C09096=1089.886,417.075,-101.948,178.028,26.123,154.162
C09097=1089.893,417.322,-101.988,178.031,26.132,154.164
C09098=1089.899,417.568,-102.030,178.035,26.142,154.166
C09099=1089.905,417.814,-102.071,178.038,26.152,154.168
C09100=1089.912,418.061,-102.112,178.042,26.162,154.170
C09101=1089.918,418.307,-102.154,178.045,26.171,154.172
C09102=1089.925,418.554,-102.196,178.048,26.181,154.174
C09103=1089.931,418.800,-102.237,178.051,26.191,154.176
C09104=1089.938,419.047,-102.278,178.055,26.201,154.179
C09105=1089.944,419.293,-102.320,178.058,26.211,154.180
C09106=1089.950,419.539,-102.361,178.062,26.221,154.183
C09107=1089.956,419.786,-102.403,178.065,26.231,154.185
C09108=1089.962,420.032,-102.444,178.069,26.241,154.187
C09109=1089.970,420.279,-102.486,178.072,26.251,154.189
C09110=1089.976,420.525,-102.527,178.075,26.261,154.191
C09111=1089.982,420.772,-102.570,178.078,26.271,154.193
C09112=1089.988,421.018,-102.611,178.082,26.281,154.195
C09113=1089.995,421.265,-102.653,178.086,26.291,154.197
C09114=1090.001,421.512,-102.695,178.089,26.302,154.200
C09115=1090.008,421.757,-102.736,178.092,26.312,154.202
C09116=1090.015,422.004,-102.778,178.096,26.322,154.204
C09117=1090.021,422.250,-102.820,178.099,26.332,154.206
C09118=1090.027,422.497,-102.861,178.103,26.343,154.208
C09119=1090.034,422.742,-102.904,178.106,26.353,154.210
C09120=1090.040,422.989,-102.945,178.110,26.364,154.213
C09121=1090.047,423.236,-102.988,178.113,26.374,154.215
C09122=1090.053,423.482,-103.029,178.117,26.385,154.217
C09123=1090.060,423.728,-103.072,178.120,26.395,154.219
C09124=1090.066,423.974,-103.113,178.124,26.406,154.221
C09125=1090.073,424.221,-103.156,178.127,26.417,154.224
C09126=1090.079,424.454,-103.196,178.130,26.427,154.226
C09127=1090.085,424.688,-103.235,178.133,26.437,154.228
C09128=1090.090,424.922,-103.276,178.137,26.447,154.230
C09129=1090.097,425.156,-103.316,178.140,26.457,154.232
C09130=1090.103,425.389,-103.356,178.144,26.467,154.235
C09131=1090.109,425.623,-103.396,178.146,26.478,154.237
C09132=1090.115,425.857,-103.436,178.150,26.488,154.239
C09133=1090.122,426.091,-103.477,178.153,26.498,154.241
C09134=1090.128,426.336,-103.519,178.157,26.509,154.244
C09135=1090.135,426.583,-103.561,178.160,26.520,154.246
C09136=1090.141,426.830,-103.604,178.163,26.531,154.248
C09137=1090.148,427.076,-103.646,178.168,26.542,154.251
C09138=1090.154,427.322,-103.688,178.171,26.553,154.253
C09139=1090.161,427.568,-103.731,178.174,26.564,154.255
C09140=1090.167,427.814,-103.774,178.178,26.575,154.258
C09141=1090.174,428.061,-103.816,178.181,26.587,154.260
C09142=1090.180,428.307,-103.859,178.185,26.597,154.262
C09143=1090.187,428.553,-103.901,178.188,26.609,154.265
C09144=1090.194,428.799,-103.944,178.192,26.620,154.267
C09145=1090.200,429.045,-103.986,178.196,26.631,154.270
C09146=1090.207,429.292,-104.030,178.199,26.643,154.272
C09147=1090.213,429.538,-104.072,178.202,26.654,154.275
C09148=1090.219,429.783,-104.116,178.206,26.665,154.277
C09149=1090.226,430.030,-104.158,178.210,26.677,154.280
C09150=1090.233,430.276,-104.201,178.213,26.688,154.282
C09151=1090.239,430.523,-104.244,178.216,26.700,154.285
C09152=1090.246,430.769,-104.286,178.220,26.712,154.287
C09153=1090.252,431.015,-104.330,178.224,26.724,154.290
C09154=1090.259,431.261,-104.373,178.227,26.735,154.292
C09155=1090.265,431.507,-104.415,178.231,26.747,154.295
C09156=1090.272,431.753,-104.459,178.235,26.759,154.297
C09157=1090.279,431.999,-104.501,178.238,26.770,154.300
C09158=1090.285,432.245,-104.545,178.241,26.782,154.302
C09159=1090.292,432.491,-104.588,178.245,26.794,154.305
C09160=1090.298,432.737,-104.632,178.249,26.806,154.308
C09161=1090.305,432.983,-104.674,178.252,26.818,154.310
C09162=1090.312,433.229,-104.718,178.255,26.830,154.313
C09163=1090.318,433.476,-104.761,178.260,26.842,154.316
C09164=1090.325,433.722,-104.804,178.263,26.854,154.318
C09165=1090.331,433.968,-104.848,178.267,26.866,154.321
C09166=1090.338,434.214,-104.891,178.270,26.879,154.324
C09167=1090.345,434.460,-104.935,178.274,26.890,154.326
C09168=1090.351,434.706,-104.978,178.278,26.903,154.329
C09169=1090.358,434.952,-105.022,178.281,26.915,154.332
C09170=1090.364,435.198,-105.065,178.284,26.927,154.334
C09171=1090.371,435.444,-105.109,178.288,26.940,154.337
C09172=1090.377,435.690,-105.153,178.292,26.952,154.340
C09173=1090.384,435.936,-105.196,178.296,26.965,154.343
C09174=1090.391,436.182,-105.240,178.299,26.977,154.345
C09175=1090.397,436.428,-105.283,178.303,26.990,154.348
C09176=1090.404,436.674,-105.327,178.306,27.002,154.351
C09177=1090.411,436.920,-105.371,178.310,27.015,154.354
C09178=1090.418,437.166,-105.415,178.314,27.028,154.356
C09179=1090.424,437.412,-105.459,178.318,27.041,154.359
C09180=1090.431,437.658,-105.503,178.321,27.053,154.362
C09181=1090.438,437.904,-105.546,178.325,27.066,154.365
C09182=1090.448,438.250,-105.608,178.330,27.084,154.369
C09183=1090.457,438.596,-105.669,178.335,27.102,154.373
C09184=1090.466,438.942,-105.732,178.340,27.121,154.377
C09185=1090.475,439.288,-105.794,178.345,27.139,154.381
C09186=1090.482,439.534,-105.838,178.349,27.152,154.384
C09187=1090.490,439.780,-105.882,178.353,27.165,154.387
C09188=1090.496,440.026,-105.926,178.356,27.178,154.390
C09189=1090.503,440.271,-105.970,178.361,27.192,154.393
C09190=1090.510,440.518,-106.015,178.364,27.205,154.396
C09191=1090.517,440.763,-106.059,178.368,27.219,154.399
C09192=1090.523,441.009,-106.103,178.372,27.232,154.402
C09193=1090.530,441.255,-106.148,178.375,27.245,154.405
C09194=1090.537,441.501,-106.192,178.379,27.259,154.408
C09195=1090.544,441.747,-106.236,178.383,27.273,154.411
C09196=1090.550,441.992,-106.281,178.386,27.286,154.414
C09197=1090.557,442.239,-106.325,178.390,27.300,154.417
C09198=1090.563,442.485,-106.370,178.394,27.313,154.420
C09199=1090.570,442.730,-106.415,178.397,27.327,154.423
C09200=1090.578,442.976,-106.460,178.401,27.341,154.427
C09201=1090.584,443.222,-106.504,178.406,27.355,154.430
C09202=1090.591,443.467,-106.548,178.410,27.369,154.433
C09203=1090.598,443.713,-106.593,178.413,27.383,154.436
C09204=1090.604,443.959,-106.638,178.417,27.397,154.439
C09205=1090.611,444.205,-106.683,178.421,27.411,154.442
C09206=1090.618,444.450,-106.728,178.425,27.425,154.446
C09207=1090.625,444.696,-106.773,178.428,27.439,154.449
C09208=1090.632,444.942,-106.817,178.431,27.453,154.452
C09209=1090.639,445.188,-106.863,178.435,27.468,154.455
C09210=1090.645,445.434,-106.907,178.438,27.481,154.459
C09211=1090.653,445.680,-106.952,178.440,27.495,154.462
C09212=1090.659,445.925,-106.997,178.443,27.509,154.465
C09213=1090.666,446.171,-107.042,178.445,27.524,154.469
C09214=1090.673,446.416,-107.088,178.447,27.538,154.472
C09215=1090.680,446.662,-107.133,178.449,27.552,154.475
C09216=1090.686,446.908,-107.178,178.452,27.566,154.479
C09217=1090.694,447.154,-107.223,178.454,27.580,154.482
C09218=1090.700,447.399,-107.269,178.455,27.593,154.485
C09219=1090.707,447.645,-107.313,178.456,27.608,154.489
C09220=1090.714,447.891,-107.359,178.458,27.622,154.492
C09221=1090.721,448.137,-107.404,178.458,27.635,154.496
C09222=1090.728,448.382,-107.450,178.459,27.649,154.499
C09223=1090.735,448.628,-107.495,178.461,27.663,154.503
C09224=1090.742,448.873,-107.540,178.461,27.677,154.506
C09225=1090.749,449.119,-107.586,178.462,27.691,154.510
C09226=1090.756,449.364,-107.631,178.462,27.705,154.513
C09227=1090.763,449.610,-107.676,178.462,27.719,154.517
C09228=1090.770,449.855,-107.721,178.463,27.732,154.520
C09229=1090.780,450.102,-107.765,178.462,27.745,154.523
C09230=1090.397,450.093,-107.952,178.418,27.943,154.578
C09231=1090.387,449.848,-107.908,178.417,27.930,154.575
C09232=1090.380,449.603,-107.862,178.417,27.917,154.571
C09233=1090.372,449.358,-107.817,178.417,27.903,154.568
C09234=1090.366,449.112,-107.771,178.416,27.889,154.564
C09235=1090.359,448.867,-107.726,178.416,27.875,154.561
C09236=1090.352,448.620,-107.680,178.415,27.861,154.557
C09237=1090.344,448.375,-107.635,178.415,27.847,154.554
C09238=1090.338,448.129,-107.590,178.413,27.833,154.550
C09239=1090.331,447.884,-107.544,178.412,27.819,154.547
C09240=1090.323,447.638,-107.499,178.411,27.805,154.543
C09241=1090.317,447.392,-107.454,178.410,27.791,154.540
C09242=1090.310,447.147,-107.408,178.407,27.777,154.537
C09243=1090.303,446.900,-107.363,178.406,27.763,154.533
C09244=1090.297,446.655,-107.318,178.404,27.749,154.530
C09245=1090.290,446.409,-107.272,178.402,27.735,154.526
C09246=1090.282,446.163,-107.227,178.399,27.721,154.523
C09247=1090.276,445.918,-107.182,178.396,27.706,154.520
C09248=1090.269,445.672,-107.137,178.394,27.692,154.516
C09249=1090.262,445.427,-107.092,178.391,27.678,154.513
C09250=1090.255,445.181,-107.047,178.388,27.664,154.510
C09251=1090.249,444.935,-107.001,178.385,27.650,154.506
C09252=1090.241,444.689,-106.957,178.380,27.636,154.503
C09253=1090.235,444.444,-106.912,178.377,27.622,154.500
C09254=1090.227,444.198,-106.867,178.373,27.607,154.497
C09255=1090.220,443.952,-106.822,178.369,27.593,154.494
C09256=1090.214,443.706,-106.777,178.366,27.580,154.490
C09257=1090.207,443.461,-106.732,178.362,27.565,154.487
C09258=1090.200,443.214,-106.687,178.358,27.551,154.484
C09259=1090.193,442.969,-106.643,178.353,27.537,154.481
C09260=1090.186,442.724,-106.598,178.350,27.524,154.478
C09261=1090.179,442.477,-106.554,178.346,27.510,154.475
C09262=1090.173,442.231,-106.509,178.342,27.496,154.472
C09263=1090.166,441.985,-106.464,178.339,27.482,154.468
C09264=1090.159,441.740,-106.419,178.335,27.468,154.465
C09265=1090.153,441.494,-106.376,178.330,27.455,154.462
C09266=1090.146,441.248,-106.331,178.327,27.442,154.459
C09267=1090.139,441.003,-106.286,178.323,27.428,154.456
C09268=1090.132,440.757,-106.242,178.320,27.415,154.453
C09269=1090.125,440.511,-106.197,178.316,27.401,154.450
C09270=1090.119,440.265,-106.153,178.312,27.387,154.447
C09271=1090.112,440.019,-106.109,178.308,27.374,154.444
C09272=1090.105,439.773,-106.065,178.304,27.361,154.441
C09273=1090.099,439.544,-106.024,178.301,27.349,154.439
C09274=1090.092,439.316,-105.982,178.297,27.337,154.436
C09275=1090.086,439.088,-105.942,178.294,27.325,154.433
C09276=1090.080,438.860,-105.901,178.290,27.312,154.430
C09277=1090.073,438.631,-105.860,178.287,27.300,154.428
C09278=1090.067,438.403,-105.819,178.284,27.288,154.425
C09279=1090.060,438.174,-105.777,178.280,27.276,154.422
C09280=1090.054,437.945,-105.738,178.276,27.264,154.420
C09281=1090.047,437.700,-105.693,178.272,27.251,154.417
C09282=1090.041,437.454,-105.649,178.268,27.238,154.414
C09283=1090.034,437.208,-105.605,178.265,27.226,154.411
C09284=1090.027,436.962,-105.562,178.262,27.213,154.408
C09285=1090.020,436.716,-105.518,178.257,27.200,154.405
C09286=1090.014,436.470,-105.474,178.254,27.188,154.403
C09287=1090.007,436.224,-105.430,178.250,27.175,154.400
C09288=1090.001,435.978,-105.386,178.247,27.163,154.397
C09289=1089.994,435.732,-105.343,178.242,27.150,154.394
C09290=1089.987,435.486,-105.299,178.239,27.138,154.392
C09291=1089.981,435.240,-105.255,178.235,27.125,154.389
C09292=1089.974,434.994,-105.212,178.231,27.113,154.386
C09293=1089.967,434.749,-105.168,178.228,27.101,154.383
C09294=1089.960,434.502,-105.124,178.224,27.088,154.381
C09295=1089.954,434.255,-105.081,178.221,27.076,154.378
C09296=1089.948,434.010,-105.038,178.217,27.064,154.375
C09297=1089.941,433.764,-104.994,178.213,27.051,154.373
C09298=1089.934,433.518,-104.950,178.210,27.039,154.370
C09299=1089.928,433.272,-104.908,178.206,27.027,154.367
C09300=1089.922,433.026,-104.864,178.202,27.015,154.365
C09301=1089.915,432.780,-104.821,178.199,27.003,154.362
C09302=1089.908,432.534,-104.778,178.195,26.991,154.359
C09303=1089.901,432.288,-104.734,178.191,26.979,154.357
C09304=1089.895,432.042,-104.691,178.188,26.967,154.354
C09305=1089.888,431.796,-104.648,178.184,26.956,154.352
C09306=1089.882,431.549,-104.605,178.180,26.943,154.349
C09307=1089.875,431.303,-104.562,178.177,26.932,154.347
C09308=1089.868,431.057,-104.518,178.173,26.920,154.344
C09309=1089.862,430.811,-104.476,178.170,26.909,154.341
C09310=1089.855,430.565,-104.432,178.165,26.897,154.339
C09311=1089.848,430.318,-104.389,178.162,26.885,154.336
C09312=1089.841,430.072,-104.347,178.159,26.874,154.334
C09313=1089.835,429.826,-104.304,178.155,26.862,154.331
C09314=1089.828,429.580,-104.261,178.151,26.851,154.329
C09315=1089.823,429.334,-104.218,178.148,26.839,154.326
C09316=1089.816,429.088,-104.175,178.144,26.828,154.324
C09317=1089.809,428.841,-104.133,178.141,26.816,154.321
C09318=1089.803,428.595,-104.090,178.137,26.805,154.319
C09319=1089.796,428.349,-104.047,178.134,26.794,154.317
C09320=1089.789,428.102,-104.004,178.130,26.782,154.314
C09321=1089.783,427.857,-103.962,178.126,26.771,154.312
C09322=1089.776,427.610,-103.920,178.123,26.760,154.309
C09323=1089.770,427.364,-103.877,178.119,26.749,154.307
C09324=1089.763,427.118,-103.834,178.116,26.738,154.305
C09325=1089.756,426.871,-103.792,178.112,26.727,154.302
C09326=1089.750,426.626,-103.749,178.109,26.716,154.300
C09327=1089.743,426.379,-103.707,178.105,26.705,154.298
C09328=1089.736,426.133,-103.664,178.101,26.694,154.295
C09329=1089.731,425.899,-103.623,178.098,26.684,154.293
C09330=1089.724,425.665,-103.584,178.095,26.673,154.291
C09331=1089.717,425.430,-103.543,178.091,26.663,154.289
C09332=1089.712,425.196,-103.503,178.088,26.653,154.286
C09333=1089.705,424.962,-103.462,178.085,26.643,154.284
C09334=1089.699,424.728,-103.423,178.081,26.632,154.282
C09335=1089.694,424.493,-103.382,178.078,26.622,154.280
C09336=1089.687,424.260,-103.342,178.074,26.612,154.278
C09337=1089.681,424.013,-103.300,178.071,26.601,154.275
C09338=1089.674,423.766,-103.258,178.067,26.591,154.273
C09339=1089.668,423.520,-103.216,178.064,26.580,154.271
C09340=1089.661,423.274,-103.174,178.060,26.569,154.269
C09341=1089.655,423.028,-103.132,178.057,26.559,154.266
C09342=1089.648,422.781,-103.090,178.053,26.548,154.264
C09343=1089.642,422.535,-103.048,178.050,26.538,154.262
C09344=1089.635,422.289,-103.006,178.046,26.527,154.260
C09345=1089.629,422.042,-102.964,178.043,26.517,154.258
C09346=1089.623,421.796,-102.922,178.040,26.507,154.256
C09347=1089.616,421.550,-102.880,178.037,26.497,154.253
C09348=1089.609,421.303,-102.838,178.033,26.487,154.251
C09349=1089.604,421.056,-102.797,178.029,26.476,154.249
C09350=1089.597,420.810,-102.754,178.026,26.466,154.247
C09351=1089.590,420.564,-102.713,178.022,26.456,154.245
C09352=1089.583,420.317,-102.671,178.019,26.446,154.243
C09353=1089.577,420.071,-102.630,178.015,26.436,154.241
C09354=1089.571,419.824,-102.588,178.012,26.426,154.238
C09355=1089.565,419.578,-102.547,178.008,26.415,154.236
C09356=1089.557,419.332,-102.505,178.005,26.406,154.234
C09357=1089.551,419.086,-102.463,178.002,26.396,154.232
C09358=1089.545,418.839,-102.421,177.998,26.386,154.230
C09359=1089.539,418.593,-102.380,177.995,26.376,154.228
C09360=1089.532,418.346,-102.339,177.991,26.366,154.226
C09361=1089.526,418.100,-102.297,177.987,26.356,154.224
C09362=1089.519,417.853,-102.255,177.985,26.346,154.222
C09363=1089.513,417.607,-102.214,177.981,26.336,154.220
C09364=1089.507,417.360,-102.174,177.978,26.327,154.218
C09365=1089.500,417.113,-102.132,177.974,26.317,154.216
C09366=1089.494,416.867,-102.091,177.970,26.307,154.214
C09367=1089.488,416.621,-102.049,177.968,26.297,154.212
C09368=1089.481,416.374,-102.008,177.964,26.288,154.210
C09369=1089.475,416.128,-101.966,177.960,26.278,154.208
C09370=1089.469,415.881,-101.925,177.957,26.268,154.206
C09371=1089.462,415.635,-101.884,177.954,26.259,154.204
C09372=1089.456,415.389,-101.843,177.950,26.250,154.202
C09373=1089.449,415.141,-101.802,177.947,26.240,154.200
C09374=1089.443,414.895,-101.761,177.943,26.230,154.198
C09375=1089.436,414.649,-101.720,177.940,26.221,154.196
C09376=1089.430,414.402,-101.679,177.937,26.212,154.194
C09377=1089.424,414.156,-101.638,177.933,26.202,154.192
C09378=1089.417,413.909,-101.598,177.930,26.194,154.190
C09379=1089.411,413.662,-101.556,177.927,26.184,154.188
C09380=1089.404,413.416,-101.516,177.923,26.175,154.187
C09381=1089.398,413.169,-101.474,177.920,26.165,154.185
C09382=1089.391,412.923,-101.434,177.917,26.156,154.183
C09383=1089.386,412.676,-101.393,177.913,26.147,154.181
C09384=1089.379,412.430,-101.352,177.910,26.138,154.179
C09385=1089.374,412.202,-101.315,177.907,26.130,154.177
C09386=1089.367,411.976,-101.277,177.903,26.121,154.176
C09387=1089.362,411.749,-101.240,177.900,26.112,154.174
C09388=1089.355,411.522,-101.203,177.897,26.105,154.172
C09389=1089.350,411.296,-101.165,177.895,26.096,154.171
C09390=1089.344,411.069,-101.128,177.892,26.088,154.169
C09391=1089.339,410.843,-101.090,177.889,26.080,154.167
C09392=1089.332,410.616,-101.053,177.886,26.072,154.165
C09393=1089.326,410.369,-101.012,177.882,26.062,154.164
C09394=1089.320,410.123,-100.972,177.878,26.053,154.162
C09395=1089.314,409.876,-100.932,177.876,26.044,154.160
C09396=1089.308,409.630,-100.891,177.872,26.036,154.158
C09397=1089.302,409.383,-100.851,177.869,26.027,154.156
C09398=1089.295,409.136,-100.810,177.865,26.018,154.155
C09399=1089.288,408.889,-100.770,177.862,26.009,154.153
C09400=1089.282,408.643,-100.729,177.859,26.000,154.151
C09401=1089.276,408.396,-100.689,177.856,25.992,154.149
C09402=1089.270,408.149,-100.649,177.852,25.983,154.148
C09403=1089.264,407.903,-100.608,177.849,25.974,154.146
C09404=1089.258,407.656,-100.568,177.846,25.965,154.144
C09405=1089.251,407.410,-100.528,177.843,25.957,154.142
C09406=1089.245,407.163,-100.488,177.839,25.948,154.141
C09407=1089.239,406.917,-100.448,177.836,25.940,154.139
C09408=1089.233,406.670,-100.407,177.832,25.931,154.137
C09409=1089.227,406.423,-100.367,177.829,25.923,154.136
C09410=1089.220,406.176,-100.327,177.826,25.914,154.134
C09411=1089.214,405.930,-100.287,177.823,25.906,154.132
C09412=1089.208,405.683,-100.247,177.820,25.897,154.130
C09413=1089.201,405.437,-100.207,177.816,25.889,154.129
C09414=1089.195,405.189,-100.168,177.813,25.881,154.127
C09415=1089.189,404.943,-100.127,177.809,25.872,154.125
C09416=1089.183,404.696,-100.087,177.807,25.864,154.124
C09417=1089.176,404.449,-100.048,177.804,25.855,154.122
C09418=1089.170,404.203,-100.008,177.800,25.847,154.121
C09419=1089.164,403.956,-99.968,177.797,25.839,154.119
C09420=1089.158,403.709,-99.928,177.793,25.830,154.117
C09421=1089.151,403.463,-99.888,177.790,25.823,154.116
C09422=1089.145,403.215,-99.849,177.787,25.814,154.114
C09423=1089.139,402.969,-99.808,177.783,25.806,154.112
C09424=1089.133,402.722,-99.769,177.781,25.798,154.111
C09425=1089.126,402.475,-99.729,177.778,25.790,154.109
C09426=1089.120,402.228,-99.689,177.774,25.782,154.108
C09427=1089.113,401.982,-99.650,177.771,25.774,154.106
C09428=1089.107,401.735,-99.610,177.768,25.766,154.104
C09429=1089.101,401.488,-99.571,177.764,25.757,154.103
C09430=1089.095,401.242,-99.531,177.761,25.749,154.101
C09431=1089.089,400.995,-99.492,177.758,25.742,154.100
C09432=1089.083,400.748,-99.452,177.754,25.734,154.098
C09433=1089.077,400.501,-99.412,177.751,25.726,154.097
C09434=1089.070,400.254,-99.373,177.748,25.718,154.095
C09435=1089.064,400.007,-99.334,177.745,25.710,154.093
C09436=1089.058,399.761,-99.294,177.742,25.702,154.092
C09437=1089.052,399.514,-99.255,177.739,25.694,154.090
C09438=1089.046,399.267,-99.215,177.736,25.686,154.089
C09439=1089.039,399.020,-99.176,177.733,25.679,154.087
C09440=1089.034,398.774,-99.137,177.729,25.671,154.086
C09441=1089.028,398.547,-99.101,177.726,25.664,154.085
C09442=1089.022,398.321,-99.065,177.723,25.656,154.083
C09443=1089.016,398.095,-99.029,177.720,25.649,154.082
C09444=1089.010,397.869,-98.994,177.717,25.642,154.080
C09445=1089.005,397.643,-98.957,177.714,25.635,154.079
C09446=1088.998,397.417,-98.921,177.712,25.629,154.078
C09447=1088.994,397.191,-98.886,177.709,25.622,154.076
C09448=1088.987,396.964,-98.850,177.706,25.614,154.075
C09449=1088.982,396.718,-98.811,177.703,25.607,154.074
C09450=1088.976,396.471,-98.772,177.700,25.599,154.072
C09451=1088.969,396.224,-98.733,177.696,25.591,154.071
C09452=1088.964,395.977,-98.694,177.692,25.584,154.069
C09453=1088.957,395.730,-98.655,177.689,25.577,154.068
C09454=1088.951,395.483,-98.616,177.686,25.569,154.066
C09455=1088.945,395.237,-98.577,177.683,25.562,154.065
C09456=1088.938,394.990,-98.538,177.680,25.554,154.063
C09457=1088.932,394.743,-98.498,177.676,25.547,154.062
C09458=1088.926,394.496,-98.461,177.673,25.539,154.061
C09459=1088.920,394.249,-98.422,177.670,25.532,154.059
C09460=1088.914,394.003,-98.383,177.667,25.525,154.058
C09461=1088.907,393.756,-98.344,177.664,25.517,154.056
C09462=1088.902,393.508,-98.305,177.661,25.510,154.055
C09463=1088.895,393.262,-98.267,177.658,25.503,154.054
C09464=1088.889,393.015,-98.227,177.654,25.495,154.052
C09465=1088.883,392.768,-98.189,177.651,25.488,154.051
C09466=1088.877,392.522,-98.151,177.648,25.480,154.050
C09467=1088.871,392.275,-98.111,177.645,25.473,154.048
C09468=1088.865,392.028,-98.073,177.642,25.466,154.047
C09469=1088.859,391.781,-98.034,177.639,25.459,154.046
C09470=1088.853,391.534,-97.996,177.636,25.452,154.044
C09471=1088.846,391.287,-97.957,177.632,25.445,154.043
C09472=1088.840,391.040,-97.920,177.629,25.438,154.042
C09473=1088.833,390.793,-97.881,177.626,25.431,154.040
C09474=1088.828,390.546,-97.842,177.622,25.424,154.039
C09475=1088.821,390.299,-97.804,177.619,25.416,154.038
C09476=1088.815,390.053,-97.766,177.616,25.409,154.036
C09477=1088.808,389.806,-97.727,177.613,25.402,154.035
C09478=1088.802,389.559,-97.689,177.610,25.396,154.034
C09479=1088.797,389.311,-97.651,177.607,25.389,154.032
C09480=1088.790,389.065,-97.612,177.604,25.382,154.031
C09481=1088.785,388.819,-97.574,177.600,25.375,154.030
C09482=1088.778,388.571,-97.536,177.597,25.368,154.028
C09483=1088.772,388.325,-97.498,177.594,25.361,154.027
C09484=1088.765,388.078,-97.460,177.591,25.354,154.026
C09485=1088.759,387.831,-97.422,177.588,25.347,154.025
C09486=1088.754,387.583,-97.383,177.585,25.340,154.023
C09487=1088.747,387.337,-97.345,177.582,25.333,154.022
C09488=1088.742,387.090,-97.307,177.578,25.327,154.021
C09489=1088.735,386.843,-97.269,177.574,25.319,154.020
C09490=1088.729,386.596,-97.231,177.571,25.313,154.018
C09491=1088.723,386.349,-97.193,177.568,25.306,154.017
C09492=1088.717,386.102,-97.155,177.565,25.299,154.016
C09493=1088.711,385.855,-97.117,177.562,25.292,154.015
C09494=1088.705,385.608,-97.080,177.558,25.286,154.013
C09495=1088.698,385.361,-97.041,177.555,25.279,154.012
C09496=1088.692,385.115,-97.003,177.552,25.272,154.011
C09497=1088.687,384.895,-96.969,177.550,25.266,154.010
C09498=1088.682,384.676,-96.936,177.547,25.260,154.009
C09499=1088.676,384.457,-96.902,177.544,25.254,154.008
C09500=1088.671,384.237,-96.868,177.542,25.248,154.007
C09501=1088.666,384.018,-96.835,177.538,25.243,154.006
C09502=1088.660,383.798,-96.801,177.536,25.237,154.005
C09503=1088.655,383.578,-96.767,177.532,25.231,154.003
C09504=1088.650,383.360,-96.734,177.530,25.225,154.002
C09505=1088.644,383.112,-96.696,177.527,25.218,154.001
C09506=1088.638,382.865,-96.659,177.524,25.212,154.000
C09507=1088.632,382.618,-96.621,177.520,25.205,153.999
C09508=1088.626,382.371,-96.583,177.517,25.198,153.998
C09509=1088.620,382.124,-96.545,177.514,25.192,153.996
C09510=1088.613,381.877,-96.508,177.511,25.186,153.995
C09511=1088.607,381.630,-96.471,177.508,25.179,153.994
C09512=1088.602,381.383,-96.433,177.505,25.173,153.993
C09513=1088.596,381.137,-96.396,177.502,25.167,153.992
C09514=1088.589,380.889,-96.358,177.499,25.160,153.991
C09515=1088.583,380.642,-96.321,177.496,25.154,153.990
C09516=1088.577,380.395,-96.283,177.492,25.148,153.988
C09517=1088.571,380.148,-96.246,177.489,25.141,153.987
C09518=1088.565,379.901,-96.208,177.486,25.135,153.986
C09519=1088.558,379.654,-96.172,177.482,25.128,153.985
C09520=1088.553,379.407,-96.134,177.479,25.122,153.984
C09521=1088.547,379.160,-96.096,177.476,25.116,153.983
C09522=1088.540,378.913,-96.060,177.474,25.110,153.982
C09523=1088.534,378.666,-96.022,177.470,25.104,153.981
C09524=1088.529,378.419,-95.985,177.467,25.097,153.979
C09525=1088.522,378.171,-95.947,177.464,25.091,153.978
C09526=1088.516,377.924,-95.910,177.461,25.085,153.977
C09527=1088.510,377.677,-95.873,177.457,25.078,153.976
C09528=1088.504,377.430,-95.836,177.454,25.072,153.975
C09529=1088.498,377.183,-95.799,177.451,25.066,153.974
C09530=1088.492,376.936,-95.761,177.448,25.060,153.973
C09531=1088.487,376.689,-95.724,177.445,25.054,153.972
C09532=1088.480,376.442,-95.688,177.442,25.047,153.971
C09533=1088.474,376.195,-95.650,177.439,25.041,153.970
C09534=1088.469,375.948,-95.613,177.435,25.035,153.969
C09535=1088.462,375.701,-95.577,177.432,25.029,153.968
C09536=1088.457,375.454,-95.540,177.430,25.023,153.966
C09537=1088.450,375.207,-95.502,177.426,25.017,153.966
C09538=1088.445,374.960,-95.465,177.423,25.011,153.964
C09539=1088.439,374.712,-95.428,177.420,25.005,153.963
C09540=1088.433,374.465,-95.392,177.416,24.999,153.962
C09541=1088.427,374.218,-95.355,177.413,24.992,153.961
C09542=1088.421,373.971,-95.318,177.411,24.987,153.960
C09543=1088.415,373.724,-95.281,177.407,24.981,153.959
C09544=1088.408,373.477,-95.244,177.404,24.975,153.958
C09545=1088.402,373.229,-95.207,177.401,24.969,153.957
C09546=1088.396,372.982,-95.170,177.397,24.963,153.956
C09547=1088.390,372.735,-95.134,177.395,24.957,153.955
C09548=1088.384,372.488,-95.097,177.392,24.951,153.954
C09549=1088.378,372.241,-95.060,177.388,24.945,153.953
C09550=1088.372,371.993,-95.023,177.385,24.939,153.952
C09551=1088.366,371.746,-94.987,177.382,24.934,153.951
C09552=1088.360,371.500,-94.951,177.379,24.928,153.950
C09553=1088.350,371.088,-94.890,177.374,24.918,153.949
C09554=1088.340,370.677,-94.829,177.368,24.908,153.947
C09555=1088.330,370.266,-94.769,177.363,24.899,153.945
C09556=1088.320,369.855,-94.708,177.358,24.889,153.944
C09557=1088.315,369.608,-94.671,177.355,24.883,153.943
C09558=1088.308,369.361,-94.635,177.352,24.878,153.942
C09559=1088.302,369.113,-94.599,177.349,24.872,153.941
C09560=1088.297,368.866,-94.562,177.345,24.866,153.940
C09561=1088.290,368.619,-94.526,177.342,24.860,153.939
C09562=1088.284,368.371,-94.490,177.339,24.855,153.938
C09563=1088.278,368.124,-94.454,177.336,24.849,153.937
C09564=1088.272,367.877,-94.416,177.333,24.844,153.936
C09565=1088.267,367.630,-94.381,177.330,24.838,153.935
C09566=1088.261,367.383,-94.345,177.327,24.832,153.934
C09567=1088.254,367.136,-94.308,177.323,24.827,153.933
C09568=1088.249,366.888,-94.272,177.320,24.821,153.932
C09569=1088.243,366.641,-94.235,177.318,24.816,153.931
C09570=1088.237,366.394,-94.200,177.314,24.810,153.930
C09571=1088.231,366.147,-94.164,177.311,24.804,153.929
C09572=1088.226,365.899,-94.127,177.308,24.799,153.928
C09573=1088.219,365.652,-94.091,177.305,24.793,153.928
C09574=1088.213,365.404,-94.055,177.302,24.787,153.927
C09575=1088.207,365.158,-94.019,177.299,24.782,153.926
C09576=1088.201,364.910,-93.983,177.296,24.776,153.925
C09577=1088.195,364.663,-93.947,177.292,24.771,153.924
C09578=1088.189,364.415,-93.911,177.290,24.766,153.923
C09579=1088.183,364.168,-93.875,177.286,24.760,153.922
C09580=1088.177,363.921,-93.839,177.283,24.755,153.921
C09581=1088.171,363.674,-93.804,177.280,24.749,153.920
C09582=1088.165,363.426,-93.768,177.277,24.743,153.919
C09583=1088.159,363.179,-93.731,177.273,24.738,153.919
C09584=1088.154,362.932,-93.696,177.271,24.733,153.918
C09585=1088.147,362.684,-93.660,177.267,24.727,153.917
C09586=1088.141,362.437,-93.625,177.264,24.722,153.916
C09587=1088.135,362.190,-93.588,177.261,24.717,153.915
C09588=1088.130,361.943,-93.553,177.258,24.711,153.914
C09589=1088.124,361.695,-93.517,177.255,24.706,153.913
C09590=1088.118,361.447,-93.481,177.252,24.701,153.913
C09591=1088.112,361.200,-93.446,177.248,24.695,153.912
C09592=1088.106,360.953,-93.410,177.245,24.690,153.911
C09593=1088.100,360.705,-93.374,177.242,24.685,153.910
C09594=1088.094,360.458,-93.338,177.239,24.679,153.909
C09595=1088.088,360.211,-93.303,177.236,24.674,153.908
C09596=1088.082,359.963,-93.267,177.233,24.669,153.907
C09597=1088.076,359.715,-93.231,177.229,24.663,153.907
C09598=1088.070,359.469,-93.197,177.227,24.658,153.906
C09599=1088.064,359.221,-93.161,177.223,24.653,153.905
C09600=1088.058,358.973,-93.125,177.221,24.648,153.904
C09601=1088.053,358.727,-93.090,177.217,24.643,153.903
C09602=1088.046,358.479,-93.055,177.214,24.638,153.902
C09603=1088.040,358.231,-93.019,177.211,24.633,153.902
C09604=1088.034,357.984,-92.983,177.208,24.627,153.901
C09605=1088.025,357.589,-92.927,177.203,24.619,153.899
C09606=1088.015,357.193,-92.871,177.198,24.611,153.898
C09607=1088.006,356.798,-92.814,177.193,24.602,153.897
C09608=1087.997,356.402,-92.758,177.188,24.594,153.896
C09609=1087.990,356.155,-92.723,177.185,24.589,153.895
C09610=1087.985,355.908,-92.688,177.182,24.584,153.894
C09611=1087.979,355.660,-92.652,177.179,24.579,153.893
C09612=1087.972,355.412,-92.617,177.176,24.574,153.892
C09613=1087.967,355.165,-92.582,177.172,24.569,153.892
C09614=1087.961,354.918,-92.546,177.170,24.564,153.891
C09615=1087.956,354.670,-92.512,177.166,24.559,153.890
C09616=1087.949,354.423,-92.477,177.163,24.553,153.889
C09617=1087.944,354.176,-92.441,177.160,24.549,153.889
C09618=1087.938,353.928,-92.406,177.157,24.544,153.888
C09619=1087.932,353.681,-92.371,177.154,24.539,153.887
C09620=1087.926,353.433,-92.336,177.150,24.534,153.886
C09621=1087.920,353.186,-92.302,177.148,24.529,153.885
C09622=1087.914,352.938,-92.266,177.144,24.523,153.885
C09623=1087.909,352.691,-92.231,177.142,24.519,153.884
C09624=1087.902,352.443,-92.196,177.138,24.514,153.883
C09625=1087.897,352.196,-92.161,177.135,24.509,153.882
C09626=1087.890,351.948,-92.126,177.132,24.504,153.882
C09627=1087.885,351.701,-92.092,177.129,24.499,153.881
C09628=1087.878,351.453,-92.057,177.126,24.494,153.880
C09629=1087.873,351.206,-92.022,177.123,24.490,153.879
C09630=1087.867,350.958,-91.987,177.120,24.484,153.879
C09631=1087.860,350.711,-91.953,177.117,24.480,153.878
C09632=1087.855,350.464,-91.918,177.113,24.475,153.877
C09633=1087.849,350.216,-91.884,177.111,24.470,153.876
C09634=1087.843,349.969,-91.848,177.107,24.465,153.876
C09635=1087.837,349.721,-91.814,177.105,24.460,153.875
C09636=1087.832,349.473,-91.779,177.101,24.455,153.874
C09637=1087.825,349.226,-91.744,177.098,24.451,153.874
C09638=1087.820,348.978,-91.709,177.095,24.445,153.873
C09639=1087.814,348.731,-91.675,177.092,24.441,153.872
C09640=1087.808,348.483,-91.641,177.088,24.436,153.871
C09641=1087.802,348.236,-91.606,177.086,24.432,153.871
C09642=1087.796,347.989,-91.572,177.082,24.426,153.870
C09643=1087.790,347.741,-91.537,177.080,24.422,153.869
C09644=1087.785,347.493,-91.502,177.076,24.417,153.869
C09645=1087.778,347.245,-91.468,177.073,24.412,153.868
C09646=1087.772,346.998,-91.434,177.071,24.408,153.867
C09647=1087.767,346.751,-91.399,177.067,24.403,153.866
C09648=1087.761,346.503,-91.364,177.064,24.398,153.866
C09649=1087.755,346.255,-91.330,177.061,24.393,153.865
C09650=1087.750,346.008,-91.296,177.058,24.389,153.864
C09651=1087.743,345.760,-91.261,177.054,24.384,153.864
C09652=1087.737,345.513,-91.227,177.052,24.379,153.863
C09653=1087.732,345.265,-91.192,177.048,24.374,153.862
C09654=1087.726,345.018,-91.158,177.045,24.370,153.862
C09655=1087.720,344.770,-91.124,177.043,24.365,153.861
C09656=1087.714,344.522,-91.090,177.039,24.361,153.860
C09657=1087.705,344.129,-91.035,177.034,24.353,153.859
C09658=1087.696,343.737,-90.982,177.029,24.346,153.858
C09659=1087.686,343.344,-90.928,177.024,24.339,153.857
C09660=1087.676,342.952,-90.873,177.020,24.332,153.856
C09661=1087.671,342.704,-90.840,177.017,24.327,153.855
C09662=1087.666,342.456,-90.805,177.013,24.322,153.855
C09663=1087.659,342.208,-90.771,177.011,24.318,153.854
C09664=1087.653,341.961,-90.737,177.008,24.314,153.853
C09665=1087.647,341.714,-90.703,177.004,24.309,153.853
C09666=1087.642,341.466,-90.669,177.001,24.304,153.852
C09667=1087.635,341.218,-90.635,176.998,24.299,153.851
C09668=1087.629,340.971,-90.601,176.995,24.295,153.851
C09669=1087.624,340.723,-90.568,176.992,24.291,153.850
C09670=1087.618,340.475,-90.533,176.989,24.286,153.849
C09671=1087.612,340.228,-90.499,176.986,24.281,153.849
C09672=1087.606,339.979,-90.466,176.983,24.277,153.848
C09673=1087.600,339.732,-90.432,176.980,24.272,153.848
C09674=1087.594,339.485,-90.398,176.977,24.268,153.847
C09675=1087.589,339.237,-90.364,176.973,24.264,153.846
C09676=1087.583,338.990,-90.330,176.971,24.259,153.846
C09677=1087.577,338.742,-90.297,176.968,24.255,153.845
C09678=1087.572,338.494,-90.263,176.964,24.250,153.844
C09679=1087.565,338.246,-90.229,176.961,24.246,153.844
C09680=1087.559,337.999,-90.195,176.959,24.242,153.843
C09681=1087.554,337.751,-90.162,176.955,24.237,153.842
C09682=1087.548,337.503,-90.128,176.952,24.233,153.842
C09683=1087.543,337.255,-90.094,176.949,24.228,153.841
C09684=1087.537,337.008,-90.060,176.946,24.224,153.841
C09685=1087.530,336.761,-90.028,176.943,24.220,153.840
C09686=1087.524,336.513,-89.993,176.940,24.215,153.839
C09687=1087.518,336.265,-89.960,176.937,24.211,153.839
C09688=1087.513,336.017,-89.926,176.934,24.206,153.838
C09689=1087.507,335.770,-89.892,176.931,24.202,153.838
C09690=1087.501,335.522,-89.859,176.927,24.198,153.837
C09691=1087.495,335.274,-89.826,176.925,24.193,153.836
C09692=1087.489,335.027,-89.792,176.922,24.189,153.836
C09693=1087.484,334.779,-89.759,176.918,24.185,153.835
C09694=1087.478,334.531,-89.726,176.915,24.180,153.835
C09695=1087.473,334.283,-89.692,176.913,24.176,153.834
C09696=1087.466,334.036,-89.659,176.910,24.172,153.833
C09697=1087.460,333.788,-89.625,176.906,24.167,153.833
C09698=1087.455,333.540,-89.592,176.903,24.163,153.832
C09699=1087.449,333.292,-89.559,176.901,24.159,153.832
C09700=1087.443,333.045,-89.526,176.897,24.154,153.831
C09701=1087.437,332.797,-89.492,176.894,24.150,153.830
C09702=1087.432,332.550,-89.459,176.891,24.146,153.830
C09703=1087.426,332.302,-89.425,176.888,24.142,153.829
C09704=1087.420,332.054,-89.393,176.885,24.137,153.829
C09705=1087.414,331.806,-89.359,176.882,24.133,153.828
C09706=1087.409,331.558,-89.326,176.879,24.129,153.828
C09707=1087.402,331.311,-89.293,176.876,24.125,153.827
C09708=1087.396,331.062,-89.259,176.873,24.121,153.826
C09709=1087.387,330.664,-89.207,176.868,24.114,153.826
C09710=1087.377,330.266,-89.154,176.863,24.107,153.825
C09711=1087.367,329.867,-89.101,176.858,24.101,153.824
C09712=1087.358,329.469,-89.047,176.853,24.095,153.823
C09713=1087.351,329.221,-89.014,176.850,24.091,153.823
C09714=1087.346,328.973,-88.981,176.847,24.086,153.822
C09715=1087.340,328.725,-88.949,176.844,24.082,153.821
C09716=1087.334,328.478,-88.917,176.841,24.078,153.821
C09717=1087.329,328.230,-88.883,176.838,24.074,153.820
C09718=1087.322,327.983,-88.850,176.835,24.070,153.820
C09719=1087.317,327.735,-88.817,176.832,24.066,153.819
C09720=1087.310,327.487,-88.784,176.829,24.062,153.819
C09721=1087.305,327.239,-88.752,176.826,24.058,153.818
C09722=1087.299,326.991,-88.719,176.822,24.054,153.818
C09723=1087.293,326.743,-88.686,176.819,24.049,153.817
C09724=1087.287,326.496,-88.653,176.817,24.045,153.817
C09725=1087.281,326.247,-88.621,176.814,24.041,153.816
C09726=1087.275,326.000,-88.588,176.811,24.037,153.815
C09727=1087.270,325.753,-88.555,176.807,24.033,153.815
C09728=1087.264,325.505,-88.522,176.804,24.029,153.815
C09729=1087.258,325.257,-88.490,176.802,24.025,153.814
C09730=1087.252,325.009,-88.457,176.799,24.021,153.813
C09731=1087.246,324.761,-88.424,176.796,24.018,153.813
C09732=1087.240,324.513,-88.392,176.792,24.013,153.812
C09733=1087.235,324.266,-88.359,176.789,24.009,153.812
C09734=1087.229,324.018,-88.327,176.786,24.005,153.811
C09735=1087.223,323.770,-88.295,176.784,24.001,153.811
C09736=1087.217,323.521,-88.262,176.781,23.997,153.810
C09737=1087.211,323.274,-88.229,176.777,23.993,153.810
C09738=1087.206,323.026,-88.198,176.774,23.989,153.809
C09739=1087.200,322.778,-88.164,176.771,23.985,153.809
C09740=1087.194,322.530,-88.132,176.768,23.981,153.808
C09741=1087.188,322.283,-88.099,176.766,23.977,153.808
C09742=1087.182,322.035,-88.068,176.763,23.974,153.807
C09743=1087.177,321.787,-88.034,176.759,23.969,153.807
C09744=1087.171,321.539,-88.002,176.756,23.965,153.806
C09745=1087.165,321.291,-87.970,176.753,23.962,153.806
C09746=1087.159,321.044,-87.938,176.750,23.957,153.805
C09747=1087.154,320.796,-87.905,176.748,23.953,153.805
C09748=1087.148,320.548,-87.873,176.745,23.950,153.804
C09749=1087.142,320.300,-87.841,176.741,23.945,153.804
C09750=1087.136,320.053,-87.808,176.738,23.941,153.803
C09751=1087.131,319.804,-87.776,176.735,23.938,153.803
C09752=1087.125,319.557,-87.744,176.732,23.934,153.802
C09753=1087.119,319.308,-87.712,176.729,23.930,153.802
C09754=1087.113,319.061,-87.679,176.727,23.926,153.801
C09755=1087.108,318.813,-87.647,176.724,23.922,153.801
C09756=1087.102,318.565,-87.615,176.720,23.918,153.800
C09757=1087.096,318.317,-87.582,176.717,23.914,153.800
C09758=1087.091,318.070,-87.551,176.714,23.910,153.799
C09759=1087.085,317.821,-87.519,176.712,23.906,153.799
C09760=1087.079,317.574,-87.487,176.709,23.902,153.798
C09761=1087.070,317.168,-87.434,176.704,23.896,153.797
C09762=1087.061,316.763,-87.382,176.698,23.890,153.797
C09763=1087.051,316.358,-87.329,176.694,23.883,153.796
C09764=1087.043,315.952,-87.277,176.689,23.877,153.795
C09765=1087.037,315.704,-87.245,176.686,23.873,153.795
C09766=1087.032,315.457,-87.213,176.683,23.869,153.794
C09767=1087.026,315.208,-87.181,176.681,23.865,153.794
C09768=1087.020,314.961,-87.149,176.678,23.862,153.793
C09769=1087.014,314.713,-87.117,176.674,23.858,153.793
C09770=1087.009,314.465,-87.086,176.671,23.854,153.792
C09771=1087.002,314.217,-87.054,176.668,23.850,153.792
C09772=1086.996,313.969,-87.022,176.665,23.846,153.791
C09773=1086.991,313.722,-86.991,176.662,23.843,153.791
C09774=1086.985,313.473,-86.959,176.659,23.839,153.790
C09775=1086.979,313.226,-86.927,176.656,23.836,153.790
C09776=1086.973,312.978,-86.895,176.654,23.832,153.789
C09777=1086.967,312.730,-86.863,176.651,23.828,153.789
C09778=1086.961,312.482,-86.832,176.648,23.824,153.789
C09779=1086.954,312.234,-86.800,176.645,23.821,153.788
C09780=1086.949,311.987,-86.769,176.641,23.817,153.788
C09781=1086.943,311.738,-86.737,176.638,23.813,153.787
C09782=1086.937,311.491,-86.706,176.635,23.810,153.787
C09783=1086.931,311.243,-86.674,176.632,23.806,153.787
C09784=1086.926,310.995,-86.643,176.629,23.802,153.786
C09785=1086.920,310.747,-86.611,176.626,23.798,153.786
C09786=1086.914,310.499,-86.580,176.623,23.795,153.785
C09787=1086.908,310.251,-86.548,176.620,23.791,153.785
C09788=1086.903,310.003,-86.517,176.617,23.787,153.784
C09789=1086.896,309.755,-86.486,176.615,23.784,153.784
C09790=1086.891,309.507,-86.454,176.612,23.780,153.784
C09791=1086.885,309.259,-86.422,176.609,23.777,153.783
C09792=1086.879,309.012,-86.391,176.606,23.773,153.783
C09793=1086.873,308.763,-86.360,176.603,23.769,153.782
C09794=1086.867,308.516,-86.329,176.599,23.765,153.782
C09795=1086.862,308.268,-86.298,176.596,23.762,153.781
C09796=1086.856,308.019,-86.266,176.593,23.758,153.781
C09797=1086.850,307.772,-86.235,176.590,23.755,153.781
C09798=1086.844,307.523,-86.203,176.587,23.751,153.780
C09799=1086.839,307.276,-86.172,176.584,23.747,153.780
C09800=1086.833,307.028,-86.141,176.581,23.744,153.779
C09801=1086.827,306.780,-86.109,176.578,23.740,153.779
C09802=1086.821,306.532,-86.079,176.575,23.737,153.778
C09803=1086.816,306.285,-86.047,176.573,23.733,153.778
C09804=1086.810,306.036,-86.016,176.570,23.729,153.778
C09805=1086.804,305.789,-85.985,176.567,23.725,153.777
C09806=1086.799,305.540,-85.954,176.564,23.722,153.777
C09807=1086.792,305.293,-85.923,176.561,23.718,153.776
C09808=1086.787,305.044,-85.892,176.558,23.714,153.776
C09809=1086.781,304.797,-85.861,176.555,23.711,153.776
C09810=1086.775,304.548,-85.829,176.552,23.708,153.775
C09811=1086.769,304.301,-85.799,176.549,23.704,153.775
C09812=1086.764,304.053,-85.767,176.546,23.701,153.774
C09813=1086.754,303.650,-85.717,176.541,23.694,153.774
C09814=1086.745,303.248,-85.667,176.537,23.689,153.773
C09815=1086.736,302.846,-85.617,176.532,23.682,153.772
C09816=1086.727,302.443,-85.566,176.527,23.677,153.772
C09817=1086.721,302.195,-85.535,176.524,23.673,153.771
C09818=1086.716,301.947,-85.505,176.521,23.670,153.771
C09819=1086.710,301.700,-85.473,176.518,23.666,153.770
C09820=1086.704,301.451,-85.443,176.515,23.663,153.770
C09821=1086.699,301.203,-85.412,176.512,23.659,153.769
C09822=1086.693,300.955,-85.381,176.510,23.655,153.769
C09823=1086.688,300.707,-85.351,176.507,23.652,153.769
C09824=1086.682,300.460,-85.319,176.504,23.648,153.768
C09825=1086.676,300.211,-85.288,176.501,23.645,153.768
C09826=1086.670,299.963,-85.258,176.498,23.641,153.767
C09827=1086.665,299.715,-85.227,176.495,23.638,153.767
C09828=1086.659,299.467,-85.196,176.492,23.634,153.767
C09829=1086.654,299.219,-85.166,176.489,23.631,153.766
C09830=1086.648,298.971,-85.135,176.486,23.627,153.766
C09831=1086.643,298.723,-85.105,176.483,23.623,153.765
C09832=1086.638,298.475,-85.074,176.480,23.620,153.765
C09833=1086.631,298.227,-85.043,176.477,23.616,153.765
C09834=1086.626,297.979,-85.012,176.474,23.612,153.764
C09835=1086.620,297.731,-84.982,176.471,23.609,153.764
C09836=1086.614,297.483,-84.952,176.468,23.606,153.764
C09837=1086.609,297.235,-84.921,176.465,23.602,153.763
C09838=1086.603,296.987,-84.891,176.463,23.598,153.763
C09839=1086.597,296.739,-84.860,176.459,23.595,153.762
C09840=1086.591,296.491,-84.829,176.456,23.592,153.762
C09841=1086.585,296.243,-84.799,176.454,23.588,153.762
C09842=1086.580,295.995,-84.768,176.450,23.585,153.761
C09843=1086.574,295.747,-84.739,176.448,23.581,153.761
C09844=1086.568,295.499,-84.708,176.445,23.578,153.760
C09845=1086.563,295.251,-84.678,176.442,23.575,153.760
C09846=1086.557,295.003,-84.647,176.439,23.571,153.760
C09847=1086.551,294.754,-84.616,176.436,23.567,153.759
C09848=1086.545,294.507,-84.586,176.433,23.564,153.759
C09849=1086.540,294.258,-84.556,176.430,23.561,153.759
C09850=1086.534,294.010,-84.526,176.428,23.558,153.758
C09851=1086.528,293.762,-84.496,176.425,23.554,153.758
C09852=1086.522,293.515,-84.465,176.422,23.551,153.757
C09853=1086.517,293.266,-84.436,176.419,23.547,153.757
C09854=1086.511,293.018,-84.405,176.416,23.544,153.757
C09855=1086.505,292.771,-84.375,176.413,23.540,153.756
C09856=1086.500,292.522,-84.345,176.410,23.537,153.756
C09857=1086.494,292.274,-84.315,176.407,23.533,153.756
C09858=1086.488,292.026,-84.285,176.404,23.530,153.755
C09859=1086.482,291.778,-84.255,176.401,23.527,153.755
C09860=1086.477,291.530,-84.225,176.398,23.524,153.755
C09861=1086.471,291.282,-84.195,176.395,23.520,153.754
C09862=1086.465,291.034,-84.165,176.392,23.516,153.754
C09863=1086.459,290.786,-84.134,176.390,23.514,153.754
C09864=1086.454,290.538,-84.105,176.387,23.510,153.753
C09865=1086.445,290.149,-84.058,176.382,23.505,153.753
C09866=1086.436,289.761,-84.011,176.377,23.499,153.752
C09867=1086.427,289.373,-83.964,176.373,23.494,153.752
C09868=1086.418,288.984,-83.917,176.368,23.489,153.751
C09869=1086.413,288.736,-83.887,176.365,23.486,153.751
C09870=1086.406,288.488,-83.858,176.362,23.482,153.750
C09871=1086.401,288.240,-83.828,176.360,23.479,153.750
C09872=1086.395,287.992,-83.798,176.357,23.476,153.750
C09873=1086.389,287.744,-83.768,176.354,23.472,153.749
C09874=1086.384,287.495,-83.738,176.351,23.469,153.749
C09875=1086.378,287.247,-83.709,176.348,23.466,153.749
C09876=1086.372,286.999,-83.679,176.345,23.462,153.748
C09877=1086.366,286.751,-83.649,176.342,23.459,153.748
C09878=1086.361,286.502,-83.619,176.339,23.456,153.748
C09879=1086.355,286.255,-83.589,176.337,23.453,153.747
C09880=1086.349,286.006,-83.560,176.334,23.449,153.747
C09881=1086.343,285.758,-83.530,176.331,23.446,153.747
C09882=1086.338,285.510,-83.501,176.328,23.442,153.746
C09883=1086.332,285.262,-83.470,176.325,23.439,153.746
C09884=1086.326,285.014,-83.442,176.322,23.436,153.745
C09885=1086.321,284.766,-83.412,176.319,23.433,153.745
C09886=1086.315,284.517,-83.382,176.316,23.429,153.745
C09887=1086.309,284.270,-83.353,176.314,23.426,153.744
C09888=1086.303,284.021,-83.323,176.311,23.423,153.744
C09889=1086.298,283.773,-83.293,176.308,23.419,153.744
C09890=1086.292,283.525,-83.264,176.305,23.416,153.744
C09891=1086.286,283.276,-83.235,176.302,23.413,153.743
C09892=1086.281,283.029,-83.205,176.299,23.409,153.743
C09893=1086.275,282.780,-83.176,176.296,23.406,153.743
C09894=1086.269,282.532,-83.147,176.294,23.403,153.742
C09895=1086.264,282.284,-83.117,176.291,23.400,153.742
C09896=1086.258,282.035,-83.087,176.288,23.397,153.742
C09897=1086.253,281.788,-83.057,176.285,23.393,153.741
C09898=1086.247,281.540,-83.028,176.282,23.390,153.741
C09899=1086.241,281.292,-82.999,176.279,23.386,153.740
C09900=1086.235,281.043,-82.970,176.277,23.384,153.740
C09901=1086.229,280.795,-82.940,176.274,23.380,153.740
C09902=1086.224,280.546,-82.911,176.271,23.377,153.739
C09903=1086.218,280.299,-82.882,176.268,23.374,153.739
C09904=1086.213,280.050,-82.853,176.265,23.370,153.739
C09905=1086.207,279.802,-82.824,176.261,23.367,153.739
C09906=1086.201,279.553,-82.794,176.259,23.364,153.738
C09907=1086.195,279.305,-82.765,176.256,23.361,153.738
C09908=1086.190,279.058,-82.736,176.253,23.358,153.738
C09909=1086.184,278.809,-82.707,176.250,23.355,153.737
C09910=1086.178,278.561,-82.677,176.247,23.351,153.737
C09911=1086.172,278.312,-82.649,176.244,23.348,153.737
C09912=1086.167,278.065,-82.620,176.242,23.345,153.736
C09913=1086.161,277.816,-82.591,176.239,23.341,153.736
C09914=1086.155,277.568,-82.561,176.236,23.338,153.736
C09915=1086.149,277.320,-82.532,176.233,23.335,153.735
C09916=1086.144,277.072,-82.504,176.230,23.332,153.735
C09917=1086.136,276.693,-82.459,176.226,23.327,153.735
C09918=1086.127,276.315,-82.415,176.222,23.322,153.734
C09919=1086.118,275.935,-82.371,176.217,23.317,153.734
C09920=1086.109,275.557,-82.327,176.213,23.312,153.733
C09921=1086.104,275.309,-82.297,176.210,23.309,153.733
C09922=1086.098,275.060,-82.269,176.208,23.306,153.732
C09923=1086.092,274.812,-82.240,176.205,23.303,153.732
C09924=1086.087,274.564,-82.210,176.202,23.300,153.732
C09925=1086.081,274.315,-82.182,176.199,23.296,153.732
C09926=1086.075,274.068,-82.153,176.196,23.293,153.731
C09927=1086.070,273.819,-82.124,176.194,23.290,153.731
C09928=1086.064,273.571,-82.095,176.191,23.287,153.731
C09929=1086.058,273.322,-82.067,176.188,23.284,153.730
C09930=1086.052,273.074,-82.038,176.185,23.281,153.730
C09931=1086.047,272.825,-82.009,176.182,23.278,153.730
C09932=1086.041,272.578,-81.981,176.179,23.275,153.729
C09933=1086.035,272.329,-81.952,176.176,23.271,153.729
C09934=1086.029,272.081,-81.923,176.173,23.268,153.729
C09935=1086.024,271.833,-81.895,176.170,23.265,153.729
C09936=1086.018,271.585,-81.866,176.168,23.262,153.728
C09937=1086.012,271.336,-81.838,176.165,23.259,153.728
C09938=1086.007,271.088,-81.809,176.162,23.256,153.728
C09939=1086.001,270.840,-81.781,176.159,23.252,153.727
C09940=1085.995,270.591,-81.752,176.157,23.249,153.727
C09941=1085.990,270.343,-81.723,176.154,23.246,153.727
C09942=1085.984,270.094,-81.695,176.151,23.243,153.726
C09943=1085.978,269.847,-81.666,176.148,23.240,153.726
C09944=1085.972,269.598,-81.638,176.146,23.237,153.726
C09945=1085.966,269.349,-81.609,176.143,23.234,153.726
C09946=1085.962,269.101,-81.581,176.140,23.231,153.725
C09947=1085.955,268.853,-81.552,176.137,23.227,153.725
C09948=1085.950,268.605,-81.524,176.135,23.224,153.725
C09949=1085.944,268.356,-81.495,176.131,23.221,153.724
C09950=1085.938,268.109,-81.467,176.128,23.218,153.724
C09951=1085.933,267.860,-81.438,176.125,23.215,153.724
C09952=1085.927,267.611,-81.410,176.123,23.212,153.723
C09953=1085.921,267.363,-81.382,176.120,23.209,153.723
C09954=1085.915,267.114,-81.354,176.117,23.206,153.723
C09955=1085.910,266.867,-81.325,176.114,23.202,153.723
C09956=1085.904,266.618,-81.297,176.112,23.200,153.722
C09957=1085.898,266.370,-81.269,176.109,23.196,153.722
C09958=1085.892,266.121,-81.241,176.106,23.193,153.722
C09959=1085.887,265.873,-81.213,176.103,23.190,153.721
C09960=1085.881,265.625,-81.184,176.101,23.187,153.721
C09961=1085.876,265.377,-81.156,176.098,23.184,153.721
C09962=1085.870,265.128,-81.128,176.095,23.180,153.720
C09963=1085.864,264.880,-81.099,176.093,23.178,153.720
C09964=1085.858,264.632,-81.071,176.090,23.175,153.720
C09965=1085.853,264.384,-81.043,176.086,23.171,153.720
C09966=1085.847,264.135,-81.015,176.083,23.168,153.719
C09967=1085.842,263.887,-80.987,176.081,23.165,153.719
C09968=1085.836,263.638,-80.958,176.078,23.162,153.719
C09969=1085.827,263.262,-80.916,176.074,23.158,153.718
C09970=1085.819,262.886,-80.874,176.070,23.153,153.718
C09971=1085.809,262.510,-80.832,176.065,23.149,153.718
C09972=1085.801,262.134,-80.790,176.061,23.144,153.717
C09973=1085.795,261.886,-80.761,176.059,23.141,153.717
C09974=1085.789,261.638,-80.734,176.055,23.138,153.717
C09975=1085.783,261.390,-80.706,176.052,23.135,153.716
C09976=1085.777,261.141,-80.678,176.050,23.132,153.716
C09977=1085.772,260.893,-80.650,176.047,23.129,153.716
C09978=1085.766,260.644,-80.622,176.044,23.126,153.716
C09979=1085.760,260.396,-80.595,176.042,23.123,153.715
C09980=1085.754,260.147,-80.567,176.039,23.120,153.715
C09981=1085.749,259.899,-80.539,176.036,23.117,153.715
C09982=1085.742,259.651,-80.511,176.034,23.114,153.714
C09983=1085.737,259.402,-80.484,176.031,23.111,153.714
C09984=1085.732,259.154,-80.456,176.028,23.108,153.714
C09985=1085.725,258.906,-80.428,176.025,23.105,153.714
C09986=1085.720,258.658,-80.400,176.022,23.102,153.713
C09987=1085.714,258.408,-80.372,176.019,23.099,153.713
C09988=1085.708,258.160,-80.345,176.016,23.096,153.713
C09989=1085.703,257.912,-80.317,176.014,23.093,153.713
C09990=1085.697,257.663,-80.289,176.011,23.090,153.712
C09991=1085.691,257.415,-80.262,176.008,23.087,153.712
C09992=1085.685,257.167,-80.234,176.006,23.084,153.712
C09993=1085.680,256.918,-80.207,176.003,23.081,153.711
C09994=1085.674,256.670,-80.179,176.000,23.077,153.711
C09995=1085.668,256.421,-80.152,175.998,23.075,153.711
C09996=1085.662,256.173,-80.124,175.995,23.072,153.711
//INST
///DATE 2021/06/17 10:54
///ATTR SC,RW,RJ
////FRAME ROBOT
///GROUP1 RB1
NOP
MOVL C00000 V=800.0 PL=0
MOVL C00001 V=800.0 PL=0
MOVL C00002 V=800.0 PL=0
MOVL C00003 V=800.0 PL=0
MOVL C00004 V=800.0 PL=0
MOVL C00005 V=800.0 PL=0
MOVL C00006 V=800.0 PL=0
MOVL C00007 V=800.0 PL=0
MOVL C00008 V=800.0 PL=0
MOVL C00009 V=800.0 PL=0
MOVL C00010 V=800.0 PL=0
MOVL C00011 V=800.0 PL=0
MOVL C00012 V=800.0 PL=0
MOVL C00013 V=800.0 PL=0
MOVL C00014 V=800.0 PL=0
MOVL C00015 V=800.0 PL=0
MOVL C00016 V=800.0 PL=0
MOVL C00017 V=800.0 PL=0
MOVL C00018 V=800.0 PL=0
MOVL C00019 V=800.0 PL=0
MOVL C00020 V=800.0 PL=0
MOVL C00021 V=800.0 PL=0
MOVL C00022 V=800.0 PL=0
MOVL C00023 V=800.0 PL=0
MOVL C00024 V=800.0 PL=0
MOVL C00025 V=800.0 PL=0
MOVL C00026 V=800.0 PL=0
MOVL C00027 V=800.0 PL=0
MOVL C00028 V=800.0 PL=0
MOVL C00029 V=800.0 PL=0
MOVL C00030 V=800.0 PL=0
MOVL C00031 V=800.0 PL=0
MOVL C00032 V=800.0 PL=0
MOVL C00033 V=800.0 PL=0
MOVL C00034 V=800.0 PL=0
MOVL C00035 V=800.0 PL=0
MOVL C00036 V=800.0 PL=0
MOVL C00037 V=800.0 PL=0
MOVL C00038 V=800.0 PL=0
MOVL C00039 V=800.0 PL=0
MOVL C00040 V=800.0 PL=0
MOVL C00041 V=800.0 PL=0
MOVL C00042 V=800.0 PL=0
MOVL C00043 V=800.0 PL=0
MOVL C00044 V=800.0 PL=0
MOVL C00045 V=800.0 PL=0
MOVL C00046 V=800.0 PL=0
MOVL C00047 V=800.0 PL=0
MOVL C00048 V=800.0 PL=0
MOVL C00049 V=800.0 PL=0
MOVL C00050 V=800.0 PL=0
MOVL C00051 V=800.0 PL=0
MOVL C00052 V=800.0 PL=0
MOVL C00053 V=800.0 PL=0
MOVL C00054 V=800.0 PL=0
MOVL C00055 V=800.0 PL=0
MOVL C00056 V=800.0 PL=0
MOVL C00057 V=800.0 PL=0
MOVL C00058 V=800.0 PL=0
MOVL C00059 V=800.0 PL=0
MOVL C00060 V=800.0 PL=0
MOVL C00061 V=800.0 PL=0
MOVL C00062 V=800.0 PL=0
MOVL C00063 V=800.0 PL=0
MOVL C00064 V=800.0 PL=0
MOVL C00065 V=800.0 PL=0
MOVL C00066 V=800.0 PL=0
MOVL C00067 V=800.0 PL=0
MOVL C00068 V=800.0 PL=0
MOVL C00069 V=800.0 PL=0
MOVL C00070 V=800.0 PL=0
MOVL C00071 V=800.0 PL=0
MOVL C00072 V=800.0 PL=0
MOVL C00073 V=800.0 PL=0
MOVL C00074 V=800.0 PL=0
MOVL C00075 V=800.0 PL=0
MOVL C00076 V=800.0 PL=0
MOVL C00077 V=800.0 PL=0
MOVL C00078 V=800.0 PL=0
MOVL C00079 V=800.0 PL=0
MOVL C00080 V=800.0 PL=0
MOVL C00081 V=800.0 PL=0
MOVL C00082 V=800.0 PL=0
MOVL C00083 V=800.0 PL=0
MOVL C00084 V=800.0 PL=0
MOVL C00085 V=800.0 PL=0
MOVL C00086 V=800.0 PL=0
MOVL C00087 V=800.0 PL=0
MOVL C00088 V=800.0 PL=0
MOVL C00089 V=800.0 PL=0
MOVL C00090 V=800.0 PL=0
MOVL C00091 V=800.0 PL=0
MOVL C00092 V=800.0 PL=0
MOVL C00093 V=800.0 PL=0
MOVL C00094 V=800.0 PL=0
MOVL C00095 V=800.0 PL=0
MOVL C00096 V=800.0 PL=0
MOVL C00097 V=800.0 PL=0
MOVL C00098 V=800.0 PL=0
MOVL C00099 V=800.0 PL=0
MOVL C00100 V=800.0 PL=0
MOVL C00101 V=800.0 PL=0
MOVL C00102 V=800.0 PL=0
MOVL C00103 V=800.0 PL=0
MOVL C00104 V=800.0 PL=0
MOVL C00105 V=800.0 PL=0
MOVL C00106 V=800.0 PL=0
MOVL C00107 V=800.0 PL=0
MOVL C00108 V=800.0 PL=0
MOVL C00109 V=800.0 PL=0
MOVL C00110 V=800.0 PL=0
MOVL C00111 V=800.0 PL=0
MOVL C00112 V=800.0 PL=0
MOVL C00113 V=800.0 PL=0
MOVL C00114 V=800.0 PL=0
MOVL C00115 V=800.0 PL=0
MOVL C00116 V=800.0 PL=0
MOVL C00117 V=800.0 PL=0
MOVL C00118 V=800.0 PL=0
MOVL C00119 V=800.0 PL=0
MOVL C00120 V=800.0 PL=0
MOVL C00121 V=800.0 PL=0
MOVL C00122 V=800.0 PL=0
MOVL C00123 V=800.0 PL=0
MOVL C00124 V=800.0 PL=0
MOVL C00125 V=800.0 PL=0
MOVL C00126 V=800.0 PL=0
MOVL C00127 V=800.0 PL=0
MOVL C00128 V=800.0 PL=0
MOVL C00129 V=800.0 PL=0
MOVL C00130 V=800.0 PL=0
MOVL C00131 V=800.0 PL=0
MOVL C00132 V=800.0 PL=0
MOVL C00133 V=800.0 PL=0
MOVL C00134 V=800.0 PL=0
MOVL C00135 V=800.0 PL=0
MOVL C00136 V=800.0 PL=0
MOVL C00137 V=800.0 PL=0
MOVL C00138 V=800.0 PL=0
MOVL C00139 V=800.0 PL=0
MOVL C00140 V=800.0 PL=0
MOVL C00141 V=800.0 PL=0
MOVL C00142 V=800.0 PL=0
MOVL C00143 V=800.0 PL=0
MOVL C00144 V=800.0 PL=0
MOVL C00145 V=800.0 PL=0
MOVL C00146 V=800.0 PL=0
MOVL C00147 V=800.0 PL=0
MOVL C00148 V=800.0 PL=0
MOVL C00149 V=800.0 PL=0
MOVL C00150 V=800.0 PL=0
MOVL C00151 V=800.0 PL=0
MOVL C00152 V=800.0 PL=0
MOVL C00153 V=800.0 PL=0
MOVL C00154 V=800.0 PL=0
MOVL C00155 V=800.0 PL=0
MOVL C00156 V=800.0 PL=0
MOVL C00157 V=800.0 PL=0
MOVL C00158 V=800.0 PL=0
MOVL C00159 V=800.0 PL=0
MOVL C00160 V=800.0 PL=0
MOVL C00161 V=800.0 PL=0
MOVL C00162 V=800.0 PL=0
MOVL C00163 V=800.0 PL=0
MOVL C00164 V=800.0 PL=0
MOVL C00165 V=800.0 PL=0
MOVL C00166 V=800.0 PL=0
MOVL C00167 V=800.0 PL=0
MOVL C00168 V=800.0 PL=0
MOVL C00169 V=800.0 PL=0
MOVL C00170 V=800.0 PL=0
MOVL C00171 V=800.0 PL=0
MOVL C00172 V=800.0 PL=0
MOVL C00173 V=800.0 PL=0
MOVL C00174 V=800.0 PL=0
MOVL C00175 V=800.0 PL=0
MOVL C00176 V=800.0 PL=0
MOVL C00177 V=800.0 PL=0
MOVL C00178 V=800.0 PL=0
MOVL C00179 V=800.0 PL=0
MOVL C00180 V=800.0 PL=0
MOVL C00181 V=800.0 PL=0
MOVL C00182 V=800.0 PL=0
MOVL C00183 V=800.0 PL=0
MOVL C00184 V=800.0 PL=0
MOVL C00185 V=800.0 PL=0
MOVL C00186 V=800.0 PL=0
MOVL C00187 V=800.0 PL=0
MOVL C00188 V=800.0 PL=0
MOVL C00189 V=800.0 PL=0
MOVL C00190 V=800.0 PL=0
MOVL C00191 V=800.0 PL=0
MOVL C00192 V=800.0 PL=0
MOVL C00193 V=800.0 PL=0
MOVL C00194 V=800.0 PL=0
MOVL C00195 V=800.0 PL=0
MOVL C00196 V=800.0 PL=0
MOVL C00197 V=800.0 PL=0
MOVL C00198 V=800.0 PL=0
MOVL C00199 V=800.0 PL=0
MOVL C00200 V=800.0 PL=0
MOVL C00201 V=800.0 PL=0
MOVL C00202 V=800.0 PL=0
MOVL C00203 V=800.0 PL=0
MOVL C00204 V=800.0 PL=0
MOVL C00205 V=800.0 PL=0
MOVL C00206 V=800.0 PL=0
MOVL C00207 V=800.0 PL=0
MOVL C00208 V=800.0 PL=0
MOVL C00209 V=800.0 PL=0
MOVL C00210 V=800.0 PL=0
MOVL C00211 V=800.0 PL=0
MOVL C00212 V=800.0 PL=0
MOVL C00213 V=800.0 PL=0
MOVL C00214 V=800.0 PL=0
MOVL C00215 V=800.0 PL=0
MOVL C00216 V=800.0 PL=0
MOVL C00217 V=800.0 PL=0
MOVL C00218 V=800.0 PL=0
MOVL C00219 V=800.0 PL=0
MOVL C00220 V=800.0 PL=0
MOVL C00221 V=800.0 PL=0
MOVL C00222 V=800.0 PL=0
MOVL C00223 V=800.0 PL=0
MOVL C00224 V=800.0 PL=0
MOVL C00225 V=800.0 PL=0
MOVL C00226 V=800.0 PL=0
MOVL C00227 V=800.0 PL=0
MOVL C00228 V=800.0 PL=0
MOVL C00229 V=800.0 PL=0
MOVL C00230 V=800.0 PL=0
MOVL C00231 V=800.0 PL=0
MOVL C00232 V=800.0 PL=0
MOVL C00233 V=800.0 PL=0
MOVL C00234 V=800.0 PL=0
MOVL C00235 V=800.0 PL=0
MOVL C00236 V=800.0 PL=0
MOVL C00237 V=800.0 PL=0
MOVL C00238 V=800.0 PL=0
MOVL C00239 V=800.0 PL=0
MOVL C00240 V=800.0 PL=0
MOVL C00241 V=800.0 PL=0
MOVL C00242 V=800.0 PL=0
MOVL C00243 V=800.0 PL=0
MOVL C00244 V=800.0 PL=0
MOVL C00245 V=800.0 PL=0
MOVL C00246 V=800.0 PL=0
MOVL C00247 V=800.0 PL=0
MOVL C00248 V=800.0 PL=0
MOVL C00249 V=800.0 PL=0
MOVL C00250 V=800.0 PL=0
MOVL C00251 V=800.0 PL=0
MOVL C00252 V=800.0 PL=0
MOVL C00253 V=800.0 PL=0
MOVL C00254 V=800.0 PL=0
MOVL C00255 V=800.0 PL=0
MOVL C00256 V=800.0 PL=0
MOVL C00257 V=800.0 PL=0
MOVL C00258 V=800.0 PL=0
MOVL C00259 V=800.0 PL=0
MOVL C00260 V=800.0 PL=0
MOVL C00261 V=800.0 PL=0
MOVL C00262 V=800.0 PL=0
MOVL C00263 V=800.0 PL=0
MOVL C00264 V=800.0 PL=0
MOVL C00265 V=800.0 PL=0
MOVL C00266 V=800.0 PL=0
MOVL C00267 V=800.0 PL=0
MOVL C00268 V=800.0 PL=0
MOVL C00269 V=800.0 PL=0
MOVL C00270 V=800.0 PL=0
MOVL C00271 V=800.0 PL=0
MOVL C00272 V=800.0 PL=0
MOVL C00273 V=800.0 PL=0
MOVL C00274 V=800.0 PL=0
MOVL C00275 V=800.0 PL=0
MOVL C00276 V=800.0 PL=0
MOVL C00277 V=800.0 PL=0
MOVL C00278 V=800.0 PL=0
MOVL C00279 V=800.0 PL=0
MOVL C00280 V=800.0 PL=0
MOVL C00281 V=800.0 PL=0
MOVL C00282 V=800.0 PL=0
MOVL C00283 V=800.0 PL=0
MOVL C00284 V=800.0 PL=0
MOVL C00285 V=800.0 PL=0
MOVL C00286 V=800.0 PL=0
MOVL C00287 V=800.0 PL=0
MOVL C00288 V=800.0 PL=0
MOVL C00289 V=800.0 PL=0
MOVL C00290 V=800.0 PL=0
MOVL C00291 V=800.0 PL=0
MOVL C00292 V=800.0 PL=0
MOVL C00293 V=800.0 PL=0
MOVL C00294 V=800.0 PL=0
MOVL C00295 V=800.0 PL=0
MOVL C00296 V=800.0 PL=0
MOVL C00297 V=800.0 PL=0
MOVL C00298 V=800.0 PL=0
MOVL C00299 V=800.0 PL=0
MOVL C00300 V=800.0 PL=0
MOVL C00301 V=800.0 PL=0
MOVL C00302 V=800.0 PL=0
MOVL C00303 V=800.0 PL=0
MOVL C00304 V=800.0 PL=0
MOVL C00305 V=800.0 PL=0
MOVL C00306 V=800.0 PL=0
MOVL C00307 V=800.0 PL=0
MOVL C00308 V=800.0 PL=0
MOVL C00309 V=800.0 PL=0
MOVL C00310 V=800.0 PL=0
MOVL C00311 V=800.0 PL=0
MOVL C00312 V=800.0 PL=0
MOVL C00313 V=800.0 PL=0
MOVL C00314 V=800.0 PL=0
MOVL C00315 V=800.0 PL=0
MOVL C00316 V=800.0 PL=0
MOVL C00317 V=800.0 PL=0
MOVL C00318 V=800.0 PL=0
MOVL C00319 V=800.0 PL=0
MOVL C00320 V=800.0 PL=0
MOVL C00321 V=800.0 PL=0
MOVL C00322 V=800.0 PL=0
MOVL C00323 V=800.0 PL=0
MOVL C00324 V=800.0 PL=0
MOVL C00325 V=800.0 PL=0
MOVL C00326 V=800.0 PL=0
MOVL C00327 V=800.0 PL=0
MOVL C00328 V=800.0 PL=0
MOVL C00329 V=800.0 PL=0
MOVL C00330 V=800.0 PL=0
MOVL C00331 V=800.0 PL=0
MOVL C00332 V=800.0 PL=0
MOVL C00333 V=800.0 PL=0
MOVL C00334 V=800.0 PL=0
MOVL C00335 V=800.0 PL=0
MOVL C00336 V=800.0 PL=0
MOVL C00337 V=800.0 PL=0
MOVL C00338 V=800.0 PL=0
MOVL C00339 V=800.0 PL=0
MOVL C00340 V=800.0 PL=0
MOVL C00341 V=800.0 PL=0
MOVL C00342 V=800.0 PL=0
MOVL C00343 V=800.0 PL=0
MOVL C00344 V=800.0 PL=0
MOVL C00345 V=800.0 PL=0
MOVL C00346 V=800.0 PL=0
MOVL C00347 V=800.0 PL=0
MOVL C00348 V=800.0 PL=0
MOVL C00349 V=800.0 PL=0
MOVL C00350 V=800.0 PL=0
MOVL C00351 V=800.0 PL=0
MOVL C00352 V=800.0 PL=0
MOVL C00353 V=800.0 PL=0
MOVL C00354 V=800.0 PL=0
MOVL C00355 V=800.0 PL=0
MOVL C00356 V=800.0 PL=0
MOVL C00357 V=800.0 PL=0
MOVL C00358 V=800.0 PL=0
MOVL C00359 V=800.0 PL=0
MOVL C00360 V=800.0 PL=0
MOVL C00361 V=800.0 PL=0
MOVL C00362 V=800.0 PL=0
MOVL C00363 V=800.0 PL=0
MOVL C00364 V=800.0 PL=0
MOVL C00365 V=800.0 PL=0
MOVL C00366 V=800.0 PL=0
MOVL C00367 V=800.0 PL=0
MOVL C00368 V=800.0 PL=0
MOVL C00369 V=800.0 PL=0
MOVL C00370 V=800.0 PL=0
MOVL C00371 V=800.0 PL=0
MOVL C00372 V=800.0 PL=0
MOVL C00373 V=800.0 PL=0
MOVL C00374 V=800.0 PL=0
MOVL C00375 V=800.0 PL=0
MOVL C00376 V=800.0 PL=0
MOVL C00377 V=800.0 PL=0
MOVL C00378 V=800.0 PL=0
MOVL C00379 V=800.0 PL=0
MOVL C00380 V=800.0 PL=0
MOVL C00381 V=800.0 PL=0
MOVL C00382 V=800.0 PL=0
MOVL C00383 V=800.0 PL=0
MOVL C00384 V=800.0 PL=0
MOVL C00385 V=800.0 PL=0
MOVL C00386 V=800.0 PL=0
MOVL C00387 V=800.0 PL=0
MOVL C00388 V=800.0 PL=0
MOVL C00389 V=800.0 PL=0
MOVL C00390 V=800.0 PL=0
MOVL C00391 V=800.0 PL=0
MOVL C00392 V=800.0 PL=0
MOVL C00393 V=800.0 PL=0
MOVL C00394 V=800.0 PL=0
MOVL C00395 V=800.0 PL=0
MOVL C00396 V=800.0 PL=0
MOVL C00397 V=800.0 PL=0
MOVL C00398 V=800.0 PL=0
MOVL C00399 V=800.0 PL=0
MOVL C00400 V=800.0 PL=0
MOVL C00401 V=800.0 PL=0
MOVL C00402 V=800.0 PL=0
MOVL C00403 V=800.0 PL=0
MOVL C00404 V=800.0 PL=0
MOVL C00405 V=800.0 PL=0
MOVL C00406 V=800.0 PL=0
MOVL C00407 V=800.0 PL=0
MOVL C00408 V=800.0 PL=0
MOVL C00409 V=800.0 PL=0
MOVL C00410 V=800.0 PL=0
MOVL C00411 V=800.0 PL=0
MOVL C00412 V=800.0 PL=0
MOVL C00413 V=800.0 PL=0
MOVL C00414 V=800.0 PL=0
MOVL C00415 V=800.0 PL=0
MOVL C00416 V=800.0 PL=0
MOVL C00417 V=800.0 PL=0
MOVL C00418 V=800.0 PL=0
MOVL C00419 V=800.0 PL=0
MOVL C00420 V=800.0 PL=0
MOVL C00421 V=800.0 PL=0
MOVL C00422 V=800.0 PL=0
MOVL C00423 V=800.0 PL=0
MOVL C00424 V=800.0 PL=0
MOVL C00425 V=800.0 PL=0
MOVL C00426 V=800.0 PL=0
MOVL C00427 V=800.0 PL=0
MOVL C00428 V=800.0 PL=0
MOVL C00429 V=800.0 PL=0
MOVL C00430 V=800.0 PL=0
MOVL C00431 V=800.0 PL=0
MOVL C00432 V=800.0 PL=0
MOVL C00433 V=800.0 PL=0
MOVL C00434 V=800.0 PL=0
MOVL C00435 V=800.0 PL=0
MOVL C00436 V=800.0 PL=0
MOVL C00437 V=800.0 PL=0
MOVL C00438 V=800.0 PL=0
MOVL C00439 V=800.0 PL=0
MOVL C00440 V=800.0 PL=0
MOVL C00441 V=800.0 PL=0
MOVL C00442 V=800.0 PL=0
MOVL C00443 V=800.0 PL=0
MOVL C00444 V=800.0 PL=0
MOVL C00445 V=800.0 PL=0
MOVL C00446 V=800.0 PL=0
MOVL C00447 V=800.0 PL=0
MOVL C00448 V=800.0 PL=0
MOVL C00449 V=800.0 PL=0
MOVL C00450 V=800.0 PL=0
MOVL C00451 V=800.0 PL=0
MOVL C00452 V=800.0 PL=0
MOVL C00453 V=800.0 PL=0
MOVL C00454 V=800.0 PL=0
MOVL C00455 V=800.0 PL=0
MOVL C00456 V=800.0 PL=0
MOVL C00457 V=800.0 PL=0
MOVL C00458 V=800.0 PL=0
MOVL C00459 V=800.0 PL=0
MOVL C00460 V=800.0 PL=0
MOVL C00461 V=800.0 PL=0
MOVL C00462 V=800.0 PL=0
MOVL C00463 V=800.0 PL=0
MOVL C00464 V=800.0 PL=0
MOVL C00465 V=800.0 PL=0
MOVL C00466 V=800.0 PL=0
MOVL C00467 V=800.0 PL=0
MOVL C00468 V=800.0 PL=0
MOVL C00469 V=800.0 PL=0
MOVL C00470 V=800.0 PL=0
MOVL C00471 V=800.0 PL=0
MOVL C00472 V=800.0 PL=0
MOVL C00473 V=800.0 PL=0
MOVL C00474 V=800.0 PL=0
MOVL C00475 V=800.0 PL=0
MOVL C00476 V=800.0 PL=0
MOVL C00477 V=800.0 PL=0
MOVL C00478 V=800.0 PL=0
MOVL C00479 V=800.0 PL=0
MOVL C00480 V=800.0 PL=0
MOVL C00481 V=800.0 PL=0
MOVL C00482 V=800.0 PL=0
MOVL C00483 V=800.0 PL=0
MOVL C00484 V=800.0 PL=0
MOVL C00485 V=800.0 PL=0
MOVL C00486 V=800.0 PL=0
MOVL C00487 V=800.0 PL=0
MOVL C00488 V=800.0 PL=0
MOVL C00489 V=800.0 PL=0
MOVL C00490 V=800.0 PL=0
MOVL C00491 V=800.0 PL=0
MOVL C00492 V=800.0 PL=0
MOVL C00493 V=800.0 PL=0
MOVL C00494 V=800.0 PL=0
MOVL C00495 V=800.0 PL=0
MOVL C00496 V=800.0 PL=0
MOVL C00497 V=800.0 PL=0
MOVL C00498 V=800.0 PL=0
MOVL C00499 V=800.0 PL=0
MOVL C00500 V=800.0 PL=0
MOVL C00501 V=800.0 PL=0
MOVL C00502 V=800.0 PL=0
MOVL C00503 V=800.0 PL=0
MOVL C00504 V=800.0 PL=0
MOVL C00505 V=800.0 PL=0
MOVL C00506 V=800.0 PL=0
MOVL C00507 V=800.0 PL=0
MOVL C00508 V=800.0 PL=0
MOVL C00509 V=800.0 PL=0
MOVL C00510 V=800.0 PL=0
MOVL C00511 V=800.0 PL=0
MOVL C00512 V=800.0 PL=0
MOVL C00513 V=800.0 PL=0
MOVL C00514 V=800.0 PL=0
MOVL C00515 V=800.0 PL=0
MOVL C00516 V=800.0 PL=0
MOVL C00517 V=800.0 PL=0
MOVL C00518 V=800.0 PL=0
MOVL C00519 V=800.0 PL=0
MOVL C00520 V=800.0 PL=0
MOVL C00521 V=800.0 PL=0
MOVL C00522 V=800.0 PL=0
MOVL C00523 V=800.0 PL=0
MOVL C00524 V=800.0 PL=0
MOVL C00525 V=800.0 PL=0
MOVL C00526 V=800.0 PL=0
MOVL C00527 V=800.0 PL=0
MOVL C00528 V=800.0 PL=0
MOVL C00529 V=800.0 PL=0
MOVL C00530 V=800.0 PL=0
MOVL C00531 V=800.0 PL=0
MOVL C00532 V=800.0 PL=0
MOVL C00533 V=800.0 PL=0
MOVL C00534 V=800.0 PL=0
MOVL C00535 V=800.0 PL=0
MOVL C00536 V=800.0 PL=0
MOVL C00537 V=800.0 PL=0
MOVL C00538 V=800.0 PL=0
MOVL C00539 V=800.0 PL=0
MOVL C00540 V=800.0 PL=0
MOVL C00541 V=800.0 PL=0
MOVL C00542 V=800.0 PL=0
MOVL C00543 V=800.0 PL=0
MOVL C00544 V=800.0 PL=0
MOVL C00545 V=800.0 PL=0
MOVL C00546 V=800.0 PL=0
MOVL C00547 V=800.0 PL=0
MOVL C00548 V=800.0 PL=0
MOVL C00549 V=800.0 PL=0
MOVL C00550 V=800.0 PL=0
MOVL C00551 V=800.0 PL=0
MOVL C00552 V=800.0 PL=0
MOVL C00553 V=800.0 PL=0
MOVL C00554 V=800.0 PL=0
MOVL C00555 V=800.0 PL=0
MOVL C00556 V=800.0 PL=0
MOVL C00557 V=800.0 PL=0
MOVL C00558 V=800.0 PL=0
MOVL C00559 V=800.0 PL=0
MOVL C00560 V=800.0 PL=0
MOVL C00561 V=800.0 PL=0
MOVL C00562 V=800.0 PL=0
MOVL C00563 V=800.0 PL=0
MOVL C00564 V=800.0 PL=0
MOVL C00565 V=800.0 PL=0
MOVL C00566 V=800.0 PL=0
MOVL C00567 V=800.0 PL=0
MOVL C00568 V=800.0 PL=0
MOVL C00569 V=800.0 PL=0
MOVL C00570 V=800.0 PL=0
MOVL C00571 V=800.0 PL=0
MOVL C00572 V=800.0 PL=0
MOVL C00573 V=800.0 PL=0
MOVL C00574 V=800.0 PL=0
MOVL C00575 V=800.0 PL=0
MOVL C00576 V=800.0 PL=0
MOVL C00577 V=800.0 PL=0
MOVL C00578 V=800.0 PL=0
MOVL C00579 V=800.0 PL=0
MOVL C00580 V=800.0 PL=0
MOVL C00581 V=800.0 PL=0
MOVL C00582 V=800.0 PL=0
MOVL C00583 V=800.0 PL=0
MOVL C00584 V=800.0 PL=0
MOVL C00585 V=800.0 PL=0
MOVL C00586 V=800.0 PL=0
MOVL C00587 V=800.0 PL=0
MOVL C00588 V=800.0 PL=0
MOVL C00589 V=800.0 PL=0
MOVL C00590 V=800.0 PL=0
MOVL C00591 V=800.0 PL=0
MOVL C00592 V=800.0 PL=0
MOVL C00593 V=800.0 PL=0
MOVL C00594 V=800.0 PL=0
MOVL C00595 V=800.0 PL=0
MOVL C00596 V=800.0 PL=0
MOVL C00597 V=800.0 PL=0
MOVL C00598 V=800.0 PL=0
MOVL C00599 V=800.0 PL=0
MOVL C00600 V=800.0 PL=0
MOVL C00601 V=800.0 PL=0
MOVL C00602 V=800.0 PL=0
MOVL C00603 V=800.0 PL=0
MOVL C00604 V=800.0 PL=0
MOVL C00605 V=800.0 PL=0
MOVL C00606 V=800.0 PL=0
MOVL C00607 V=800.0 PL=0
MOVL C00608 V=800.0 PL=0
MOVL C00609 V=800.0 PL=0
MOVL C00610 V=800.0 PL=0
MOVL C00611 V=800.0 PL=0
MOVL C00612 V=800.0 PL=0
MOVL C00613 V=800.0 PL=0
MOVL C00614 V=800.0 PL=0
MOVL C00615 V=800.0 PL=0
MOVL C00616 V=800.0 PL=0
MOVL C00617 V=800.0 PL=0
MOVL C00618 V=800.0 PL=0
MOVL C00619 V=800.0 PL=0
MOVL C00620 V=800.0 PL=0
MOVL C00621 V=800.0 PL=0
MOVL C00622 V=800.0 PL=0
MOVL C00623 V=800.0 PL=0
MOVL C00624 V=800.0 PL=0
MOVL C00625 V=800.0 PL=0
MOVL C00626 V=800.0 PL=0
MOVL C00627 V=800.0 PL=0
MOVL C00628 V=800.0 PL=0
MOVL C00629 V=800.0 PL=0
MOVL C00630 V=800.0 PL=0
MOVL C00631 V=800.0 PL=0
MOVL C00632 V=800.0 PL=0
MOVL C00633 V=800.0 PL=0
MOVL C00634 V=800.0 PL=0
MOVL C00635 V=800.0 PL=0
MOVL C00636 V=800.0 PL=0
MOVL C00637 V=800.0 PL=0
MOVL C00638 V=800.0 PL=0
MOVL C00639 V=800.0 PL=0
MOVL C00640 V=800.0 PL=0
MOVL C00641 V=800.0 PL=0
MOVL C00642 V=800.0 PL=0
MOVL C00643 V=800.0 PL=0
MOVL C00644 V=800.0 PL=0
MOVL C00645 V=800.0 PL=0
MOVL C00646 V=800.0 PL=0
MOVL C00647 V=800.0 PL=0
MOVL C00648 V=800.0 PL=0
MOVL C00649 V=800.0 PL=0
MOVL C00650 V=800.0 PL=0
MOVL C00651 V=800.0 PL=0
MOVL C00652 V=800.0 PL=0
MOVL C00653 V=800.0 PL=0
MOVL C00654 V=800.0 PL=0
MOVL C00655 V=800.0 PL=0
MOVL C00656 V=800.0 PL=0
MOVL C00657 V=800.0 PL=0
MOVL C00658 V=800.0 PL=0
MOVL C00659 V=800.0 PL=0
MOVL C00660 V=800.0 PL=0
MOVL C00661 V=800.0 PL=0
MOVL C00662 V=800.0 PL=0
MOVL C00663 V=800.0 PL=0
MOVL C00664 V=800.0 PL=0
MOVL C00665 V=800.0 PL=0
MOVL C00666 V=800.0 PL=0
MOVL C00667 V=800.0 PL=0
MOVL C00668 V=800.0 PL=0
MOVL C00669 V=800.0 PL=0
MOVL C00670 V=800.0 PL=0
MOVL C00671 V=800.0 PL=0
MOVL C00672 V=800.0 PL=0
MOVL C00673 V=800.0 PL=0
MOVL C00674 V=800.0 PL=0
MOVL C00675 V=800.0 PL=0
MOVL C00676 V=800.0 PL=0
MOVL C00677 V=800.0 PL=0
MOVL C00678 V=800.0 PL=0
MOVL C00679 V=800.0 PL=0
MOVL C00680 V=800.0 PL=0
MOVL C00681 V=800.0 PL=0
MOVL C00682 V=800.0 PL=0
MOVL C00683 V=800.0 PL=0
MOVL C00684 V=800.0 PL=0
MOVL C00685 V=800.0 PL=0
MOVL C00686 V=800.0 PL=0
MOVL C00687 V=800.0 PL=0
MOVL C00688 V=800.0 PL=0
MOVL C00689 V=800.0 PL=0
MOVL C00690 V=800.0 PL=0
MOVL C00691 V=800.0 PL=0
MOVL C00692 V=800.0 PL=0
MOVL C00693 V=800.0 PL=0
MOVL C00694 V=800.0 PL=0
MOVL C00695 V=800.0 PL=0
MOVL C00696 V=800.0 PL=0
MOVL C00697 V=800.0 PL=0
MOVL C00698 V=800.0 PL=0
MOVL C00699 V=800.0 PL=0
MOVL C00700 V=800.0 PL=0
MOVL C00701 V=800.0 PL=0
MOVL C00702 V=800.0 PL=0
MOVL C00703 V=800.0 PL=0
MOVL C00704 V=800.0 PL=0
MOVL C00705 V=800.0 PL=0
MOVL C00706 V=800.0 PL=0
MOVL C00707 V=800.0 PL=0
MOVL C00708 V=800.0 PL=0
MOVL C00709 V=800.0 PL=0
MOVL C00710 V=800.0 PL=0
MOVL C00711 V=800.0 PL=0
MOVL C00712 V=800.0 PL=0
MOVL C00713 V=800.0 PL=0
MOVL C00714 V=800.0 PL=0
MOVL C00715 V=800.0 PL=0
MOVL C00716 V=800.0 PL=0
MOVL C00717 V=800.0 PL=0
MOVL C00718 V=800.0 PL=0
MOVL C00719 V=800.0 PL=0
MOVL C00720 V=800.0 PL=0
MOVL C00721 V=800.0 PL=0
MOVL C00722 V=800.0 PL=0
MOVL C00723 V=800.0 PL=0
MOVL C00724 V=800.0 PL=0
MOVL C00725 V=800.0 PL=0
MOVL C00726 V=800.0 PL=0
MOVL C00727 V=800.0 PL=0
MOVL C00728 V=800.0 PL=0
MOVL C00729 V=800.0 PL=0
MOVL C00730 V=800.0 PL=0
MOVL C00731 V=800.0 PL=0
MOVL C00732 V=800.0 PL=0
MOVL C00733 V=800.0 PL=0
MOVL C00734 V=800.0 PL=0
MOVL C00735 V=800.0 PL=0
MOVL C00736 V=800.0 PL=0
MOVL C00737 V=800.0 PL=0
MOVL C00738 V=800.0 PL=0
MOVL C00739 V=800.0 PL=0
MOVL C00740 V=800.0 PL=0
MOVL C00741 V=800.0 PL=0
MOVL C00742 V=800.0 PL=0
MOVL C00743 V=800.0 PL=0
MOVL C00744 V=800.0 PL=0
MOVL C00745 V=800.0 PL=0
MOVL C00746 V=800.0 PL=0
MOVL C00747 V=800.0 PL=0
MOVL C00748 V=800.0 PL=0
MOVL C00749 V=800.0 PL=0
MOVL C00750 V=800.0 PL=0
MOVL C00751 V=800.0 PL=0
MOVL C00752 V=800.0 PL=0
MOVL C00753 V=800.0 PL=0
MOVL C00754 V=800.0 PL=0
MOVL C00755 V=800.0 PL=0
MOVL C00756 V=800.0 PL=0
MOVL C00757 V=800.0 PL=0
MOVL C00758 V=800.0 PL=0
MOVL C00759 V=800.0 PL=0
MOVL C00760 V=800.0 PL=0
MOVL C00761 V=800.0 PL=0
MOVL C00762 V=800.0 PL=0
MOVL C00763 V=800.0 PL=0
MOVL C00764 V=800.0 PL=0
MOVL C00765 V=800.0 PL=0
MOVL C00766 V=800.0 PL=0
MOVL C00767 V=800.0 PL=0
MOVL C00768 V=800.0 PL=0
MOVL C00769 V=800.0 PL=0
MOVL C00770 V=800.0 PL=0
MOVL C00771 V=800.0 PL=0
MOVL C00772 V=800.0 PL=0
MOVL C00773 V=800.0 PL=0
MOVL C00774 V=800.0 PL=0
MOVL C00775 V=800.0 PL=0
MOVL C00776 V=800.0 PL=0
MOVL C00777 V=800.0 PL=0
MOVL C00778 V=800.0 PL=0
MOVL C00779 V=800.0 PL=0
MOVL C00780 V=800.0 PL=0
MOVL C00781 V=800.0 PL=0
MOVL C00782 V=800.0 PL=0
MOVL C00783 V=800.0 PL=0
MOVL C00784 V=800.0 PL=0
MOVL C00785 V=800.0 PL=0
MOVL C00786 V=800.0 PL=0
MOVL C00787 V=800.0 PL=0
MOVL C00788 V=800.0 PL=0
MOVL C00789 V=800.0 PL=0
MOVL C00790 V=800.0 PL=0
MOVL C00791 V=800.0 PL=0
MOVL C00792 V=800.0 PL=0
MOVL C00793 V=800.0 PL=0
MOVL C00794 V=800.0 PL=0
MOVL C00795 V=800.0 PL=0
MOVL C00796 V=800.0 PL=0
MOVL C00797 V=800.0 PL=0
MOVL C00798 V=800.0 PL=0
MOVL C00799 V=800.0 PL=0
MOVL C00800 V=800.0 PL=0
MOVL C00801 V=800.0 PL=0
MOVL C00802 V=800.0 PL=0
MOVL C00803 V=800.0 PL=0
MOVL C00804 V=800.0 PL=0
MOVL C00805 V=800.0 PL=0
MOVL C00806 V=800.0 PL=0
MOVL C00807 V=800.0 PL=0
MOVL C00808 V=800.0 PL=0
MOVL C00809 V=800.0 PL=0
MOVL C00810 V=800.0 PL=0
MOVL C00811 V=800.0 PL=0
MOVL C00812 V=800.0 PL=0
MOVL C00813 V=800.0 PL=0
MOVL C00814 V=800.0 PL=0
MOVL C00815 V=800.0 PL=0
MOVL C00816 V=800.0 PL=0
MOVL C00817 V=800.0 PL=0
MOVL C00818 V=800.0 PL=0
MOVL C00819 V=800.0 PL=0
MOVL C00820 V=800.0 PL=0
MOVL C00821 V=800.0 PL=0
MOVL C00822 V=800.0 PL=0
MOVL C00823 V=800.0 PL=0
MOVL C00824 V=800.0 PL=0
MOVL C00825 V=800.0 PL=0
MOVL C00826 V=800.0 PL=0
MOVL C00827 V=800.0 PL=0
MOVL C00828 V=800.0 PL=0
MOVL C00829 V=800.0 PL=0
MOVL C00830 V=800.0 PL=0
MOVL C00831 V=800.0 PL=0
MOVL C00832 V=800.0 PL=0
MOVL C00833 V=800.0 PL=0
MOVL C00834 V=800.0 PL=0
MOVL C00835 V=800.0 PL=0
MOVL C00836 V=800.0 PL=0
MOVL C00837 V=800.0 PL=0
MOVL C00838 V=800.0 PL=0
MOVL C00839 V=800.0 PL=0
MOVL C00840 V=800.0 PL=0
MOVL C00841 V=800.0 PL=0
MOVL C00842 V=800.0 PL=0
MOVL C00843 V=800.0 PL=0
MOVL C00844 V=800.0 PL=0
MOVL C00845 V=800.0 PL=0
MOVL C00846 V=800.0 PL=0
MOVL C00847 V=800.0 PL=0
MOVL C00848 V=800.0 PL=0
MOVL C00849 V=800.0 PL=0
MOVL C00850 V=800.0 PL=0
MOVL C00851 V=800.0 PL=0
MOVL C00852 V=800.0 PL=0
MOVL C00853 V=800.0 PL=0
MOVL C00854 V=800.0 PL=0
MOVL C00855 V=800.0 PL=0
MOVL C00856 V=800.0 PL=0
MOVL C00857 V=800.0 PL=0
MOVL C00858 V=800.0 PL=0
MOVL C00859 V=800.0 PL=0
MOVL C00860 V=800.0 PL=0
MOVL C00861 V=800.0 PL=0
MOVL C00862 V=800.0 PL=0
MOVL C00863 V=800.0 PL=0
MOVL C00864 V=800.0 PL=0
MOVL C00865 V=800.0 PL=0
MOVL C00866 V=800.0 PL=0
MOVL C00867 V=800.0 PL=0
MOVL C00868 V=800.0 PL=0
MOVL C00869 V=800.0 PL=0
MOVL C00870 V=800.0 PL=0
MOVL C00871 V=800.0 PL=0
MOVL C00872 V=800.0 PL=0
MOVL C00873 V=800.0 PL=0
MOVL C00874 V=800.0 PL=0
MOVL C00875 V=800.0 PL=0
MOVL C00876 V=800.0 PL=0
MOVL C00877 V=800.0 PL=0
MOVL C00878 V=800.0 PL=0
MOVL C00879 V=800.0 PL=0
MOVL C00880 V=800.0 PL=0
MOVL C00881 V=800.0 PL=0
MOVL C00882 V=800.0 PL=0
MOVL C00883 V=800.0 PL=0
MOVL C00884 V=800.0 PL=0
MOVL C00885 V=800.0 PL=0
MOVL C00886 V=800.0 PL=0
MOVL C00887 V=800.0 PL=0
MOVL C00888 V=800.0 PL=0
MOVL C00889 V=800.0 PL=0
MOVL C00890 V=800.0 PL=0
MOVL C00891 V=800.0 PL=0
MOVL C00892 V=800.0 PL=0
MOVL C00893 V=800.0 PL=0
MOVL C00894 V=800.0 PL=0
MOVL C00895 V=800.0 PL=0
MOVL C00896 V=800.0 PL=0
MOVL C00897 V=800.0 PL=0
MOVL C00898 V=800.0 PL=0
MOVL C00899 V=800.0 PL=0
MOVL C00900 V=800.0 PL=0
MOVL C00901 V=800.0 PL=0
MOVL C00902 V=800.0 PL=0
MOVL C00903 V=800.0 PL=0
MOVL C00904 V=800.0 PL=0
MOVL C00905 V=800.0 PL=0
MOVL C00906 V=800.0 PL=0
MOVL C00907 V=800.0 PL=0
MOVL C00908 V=800.0 PL=0
MOVL C00909 V=800.0 PL=0
MOVL C00910 V=800.0 PL=0
MOVL C00911 V=800.0 PL=0
MOVL C00912 V=800.0 PL=0
MOVL C00913 V=800.0 PL=0
MOVL C00914 V=800.0 PL=0
MOVL C00915 V=800.0 PL=0
MOVL C00916 V=800.0 PL=0
MOVL C00917 V=800.0 PL=0
MOVL C00918 V=800.0 PL=0
MOVL C00919 V=800.0 PL=0
MOVL C00920 V=800.0 PL=0
MOVL C00921 V=800.0 PL=0
MOVL C00922 V=800.0 PL=0
MOVL C00923 V=800.0 PL=0
MOVL C00924 V=800.0 PL=0
MOVL C00925 V=800.0 PL=0
MOVL C00926 V=800.0 PL=0
MOVL C00927 V=800.0 PL=0
MOVL C00928 V=800.0 PL=0
MOVL C00929 V=800.0 PL=0
MOVL C00930 V=800.0 PL=0
MOVL C00931 V=800.0 PL=0
MOVL C00932 V=800.0 PL=0
MOVL C00933 V=800.0 PL=0
MOVL C00934 V=800.0 PL=0
MOVL C00935 V=800.0 PL=0
MOVL C00936 V=800.0 PL=0
MOVL C00937 V=800.0 PL=0
MOVL C00938 V=800.0 PL=0
MOVL C00939 V=800.0 PL=0
MOVL C00940 V=800.0 PL=0
MOVL C00941 V=800.0 PL=0
MOVL C00942 V=800.0 PL=0
MOVL C00943 V=800.0 PL=0
MOVL C00944 V=800.0 PL=0
MOVL C00945 V=800.0 PL=0
MOVL C00946 V=800.0 PL=0
MOVL C00947 V=800.0 PL=0
MOVL C00948 V=800.0 PL=0
MOVL C00949 V=800.0 PL=0
MOVL C00950 V=800.0 PL=0
MOVL C00951 V=800.0 PL=0
MOVL C00952 V=800.0 PL=0
MOVL C00953 V=800.0 PL=0
MOVL C00954 V=800.0 PL=0
MOVL C00955 V=800.0 PL=0
MOVL C00956 V=800.0 PL=0
MOVL C00957 V=800.0 PL=0
MOVL C00958 V=800.0 PL=0
MOVL C00959 V=800.0 PL=0
MOVL C00960 V=800.0 PL=0
MOVL C00961 V=800.0 PL=0
MOVL C00962 V=800.0 PL=0
MOVL C00963 V=800.0 PL=0
MOVL C00964 V=800.0 PL=0
MOVL C00965 V=800.0 PL=0
MOVL C00966 V=800.0 PL=0
MOVL C00967 V=800.0 PL=0
MOVL C00968 V=800.0 PL=0
MOVL C00969 V=800.0 PL=0
MOVL C00970 V=800.0 PL=0
MOVL C00971 V=800.0 PL=0
MOVL C00972 V=800.0 PL=0
MOVL C00973 V=800.0 PL=0
MOVL C00974 V=800.0 PL=0
MOVL C00975 V=800.0 PL=0
MOVL C00976 V=800.0 PL=0
MOVL C00977 V=800.0 PL=0
MOVL C00978 V=800.0 PL=0
MOVL C00979 V=800.0 PL=0
MOVL C00980 V=800.0 PL=0
MOVL C00981 V=800.0 PL=0
MOVL C00982 V=800.0 PL=0
MOVL C00983 V=800.0 PL=0
MOVL C00984 V=800.0 PL=0
MOVL C00985 V=800.0 PL=0
MOVL C00986 V=800.0 PL=0
MOVL C00987 V=800.0 PL=0
MOVL C00988 V=800.0 PL=0
MOVL C00989 V=800.0 PL=0
MOVL C00990 V=800.0 PL=0
MOVL C00991 V=800.0 PL=0
MOVL C00992 V=800.0 PL=0
MOVL C00993 V=800.0 PL=0
MOVL C00994 V=800.0 PL=0
MOVL C00995 V=800.0 PL=0
MOVL C00996 V=800.0 PL=0
MOVL C00997 V=800.0 PL=0
MOVL C00998 V=800.0 PL=0
MOVL C00999 V=800.0 PL=0
MOVL C01000 V=800.0 PL=0
MOVL C01001 V=800.0 PL=0
MOVL C01002 V=800.0 PL=0
MOVL C01003 V=800.0 PL=0
MOVL C01004 V=800.0 PL=0
MOVL C01005 V=800.0 PL=0
MOVL C01006 V=800.0 PL=0
MOVL C01007 V=800.0 PL=0
MOVL C01008 V=800.0 PL=0
MOVL C01009 V=800.0 PL=0
MOVL C01010 V=800.0 PL=0
MOVL C01011 V=800.0 PL=0
MOVL C01012 V=800.0 PL=0
MOVL C01013 V=800.0 PL=0
MOVL C01014 V=800.0 PL=0
MOVL C01015 V=800.0 PL=0
MOVL C01016 V=800.0 PL=0
MOVL C01017 V=800.0 PL=0
MOVL C01018 V=800.0 PL=0
MOVL C01019 V=800.0 PL=0
MOVL C01020 V=800.0 PL=0
MOVL C01021 V=800.0 PL=0
MOVL C01022 V=800.0 PL=0
MOVL C01023 V=800.0 PL=0
MOVL C01024 V=800.0 PL=0
MOVL C01025 V=800.0 PL=0
MOVL C01026 V=800.0 PL=0
MOVL C01027 V=800.0 PL=0
MOVL C01028 V=800.0 PL=0
MOVL C01029 V=800.0 PL=0
MOVL C01030 V=800.0 PL=0
MOVL C01031 V=800.0 PL=0
MOVL C01032 V=800.0 PL=0
MOVL C01033 V=800.0 PL=0
MOVL C01034 V=800.0 PL=0
MOVL C01035 V=800.0 PL=0
MOVL C01036 V=800.0 PL=0
MOVL C01037 V=800.0 PL=0
MOVL C01038 V=800.0 PL=0
MOVL C01039 V=800.0 PL=0
MOVL C01040 V=800.0 PL=0
MOVL C01041 V=800.0 PL=0
MOVL C01042 V=800.0 PL=0
MOVL C01043 V=800.0 PL=0
MOVL C01044 V=800.0 PL=0
MOVL C01045 V=800.0 PL=0
MOVL C01046 V=800.0 PL=0
MOVL C01047 V=800.0 PL=0
MOVL C01048 V=800.0 PL=0
MOVL C01049 V=800.0 PL=0
MOVL C01050 V=800.0 PL=0
MOVL C01051 V=800.0 PL=0
MOVL C01052 V=800.0 PL=0
MOVL C01053 V=800.0 PL=0
MOVL C01054 V=800.0 PL=0
MOVL C01055 V=800.0 PL=0
MOVL C01056 V=800.0 PL=0
MOVL C01057 V=800.0 PL=0
MOVL C01058 V=800.0 PL=0
MOVL C01059 V=800.0 PL=0
MOVL C01060 V=800.0 PL=0
MOVL C01061 V=800.0 PL=0
MOVL C01062 V=800.0 PL=0
MOVL C01063 V=800.0 PL=0
MOVL C01064 V=800.0 PL=0
MOVL C01065 V=800.0 PL=0
MOVL C01066 V=800.0 PL=0
MOVL C01067 V=800.0 PL=0
MOVL C01068 V=800.0 PL=0
MOVL C01069 V=800.0 PL=0
MOVL C01070 V=800.0 PL=0
MOVL C01071 V=800.0 PL=0
MOVL C01072 V=800.0 PL=0
MOVL C01073 V=800.0 PL=0
MOVL C01074 V=800.0 PL=0
MOVL C01075 V=800.0 PL=0
MOVL C01076 V=800.0 PL=0
MOVL C01077 V=800.0 PL=0
MOVL C01078 V=800.0 PL=0
MOVL C01079 V=800.0 PL=0
MOVL C01080 V=800.0 PL=0
MOVL C01081 V=800.0 PL=0
MOVL C01082 V=800.0 PL=0
MOVL C01083 V=800.0 PL=0
MOVL C01084 V=800.0 PL=0
MOVL C01085 V=800.0 PL=0
MOVL C01086 V=800.0 PL=0
MOVL C01087 V=800.0 PL=0
MOVL C01088 V=800.0 PL=0
MOVL C01089 V=800.0 PL=0
MOVL C01090 V=800.0 PL=0
MOVL C01091 V=800.0 PL=0
MOVL C01092 V=800.0 PL=0
MOVL C01093 V=800.0 PL=0
MOVL C01094 V=800.0 PL=0
MOVL C01095 V=800.0 PL=0
MOVL C01096 V=800.0 PL=0
MOVL C01097 V=800.0 PL=0
MOVL C01098 V=800.0 PL=0
MOVL C01099 V=800.0 PL=0
MOVL C01100 V=800.0 PL=0
MOVL C01101 V=800.0 PL=0
MOVL C01102 V=800.0 PL=0
MOVL C01103 V=800.0 PL=0
MOVL C01104 V=800.0 PL=0
MOVL C01105 V=800.0 PL=0
MOVL C01106 V=800.0 PL=0
MOVL C01107 V=800.0 PL=0
MOVL C01108 V=800.0 PL=0
MOVL C01109 V=800.0 PL=0
MOVL C01110 V=800.0 PL=0
MOVL C01111 V=800.0 PL=0
MOVL C01112 V=800.0 PL=0
MOVL C01113 V=800.0 PL=0
MOVL C01114 V=800.0 PL=0
MOVL C01115 V=800.0 PL=0
MOVL C01116 V=800.0 PL=0
MOVL C01117 V=800.0 PL=0
MOVL C01118 V=800.0 PL=0
MOVL C01119 V=800.0 PL=0
MOVL C01120 V=800.0 PL=0
MOVL C01121 V=800.0 PL=0
MOVL C01122 V=800.0 PL=0
MOVL C01123 V=800.0 PL=0
MOVL C01124 V=800.0 PL=0
MOVL C01125 V=800.0 PL=0
MOVL C01126 V=800.0 PL=0
MOVL C01127 V=800.0 PL=0
MOVL C01128 V=800.0 PL=0
MOVL C01129 V=800.0 PL=0
MOVL C01130 V=800.0 PL=0
MOVL C01131 V=800.0 PL=0
MOVL C01132 V=800.0 PL=0
MOVL C01133 V=800.0 PL=0
MOVL C01134 V=800.0 PL=0
MOVL C01135 V=800.0 PL=0
MOVL C01136 V=800.0 PL=0
MOVL C01137 V=800.0 PL=0
MOVL C01138 V=800.0 PL=0
MOVL C01139 V=800.0 PL=0
MOVL C01140 V=800.0 PL=0
MOVL C01141 V=800.0 PL=0
MOVL C01142 V=800.0 PL=0
MOVL C01143 V=800.0 PL=0
MOVL C01144 V=800.0 PL=0
MOVL C01145 V=800.0 PL=0
MOVL C01146 V=800.0 PL=0
MOVL C01147 V=800.0 PL=0
MOVL C01148 V=800.0 PL=0
MOVL C01149 V=800.0 PL=0
MOVL C01150 V=800.0 PL=0
MOVL C01151 V=800.0 PL=0
MOVL C01152 V=800.0 PL=0
MOVL C01153 V=800.0 PL=0
MOVL C01154 V=800.0 PL=0
MOVL C01155 V=800.0 PL=0
MOVL C01156 V=800.0 PL=0
MOVL C01157 V=800.0 PL=0
MOVL C01158 V=800.0 PL=0
MOVL C01159 V=800.0 PL=0
MOVL C01160 V=800.0 PL=0
MOVL C01161 V=800.0 PL=0
MOVL C01162 V=800.0 PL=0
MOVL C01163 V=800.0 PL=0
MOVL C01164 V=800.0 PL=0
MOVL C01165 V=800.0 PL=0
MOVL C01166 V=800.0 PL=0
MOVL C01167 V=800.0 PL=0
MOVL C01168 V=800.0 PL=0
MOVL C01169 V=800.0 PL=0
MOVL C01170 V=800.0 PL=0
MOVL C01171 V=800.0 PL=0
MOVL C01172 V=800.0 PL=0
MOVL C01173 V=800.0 PL=0
MOVL C01174 V=800.0 PL=0
MOVL C01175 V=800.0 PL=0
MOVL C01176 V=800.0 PL=0
MOVL C01177 V=800.0 PL=0
MOVL C01178 V=800.0 PL=0
MOVL C01179 V=800.0 PL=0
MOVL C01180 V=800.0 PL=0
MOVL C01181 V=800.0 PL=0
MOVL C01182 V=800.0 PL=0
MOVL C01183 V=800.0 PL=0
MOVL C01184 V=800.0 PL=0
MOVL C01185 V=800.0 PL=0
MOVL C01186 V=800.0 PL=0
MOVL C01187 V=800.0 PL=0
MOVL C01188 V=800.0 PL=0
MOVL C01189 V=800.0 PL=0
MOVL C01190 V=800.0 PL=0
MOVL C01191 V=800.0 PL=0
MOVL C01192 V=800.0 PL=0
MOVL C01193 V=800.0 PL=0
MOVL C01194 V=800.0 PL=0
MOVL C01195 V=800.0 PL=0
MOVL C01196 V=800.0 PL=0
MOVL C01197 V=800.0 PL=0
MOVL C01198 V=800.0 PL=0
MOVL C01199 V=800.0 PL=0
MOVL C01200 V=800.0 PL=0
MOVL C01201 V=800.0 PL=0
MOVL C01202 V=800.0 PL=0
MOVL C01203 V=800.0 PL=0
MOVL C01204 V=800.0 PL=0
MOVL C01205 V=800.0 PL=0
MOVL C01206 V=800.0 PL=0
MOVL C01207 V=800.0 PL=0
MOVL C01208 V=800.0 PL=0
MOVL C01209 V=800.0 PL=0
MOVL C01210 V=800.0 PL=0
MOVL C01211 V=800.0 PL=0
MOVL C01212 V=800.0 PL=0
MOVL C01213 V=800.0 PL=0
MOVL C01214 V=800.0 PL=0
MOVL C01215 V=800.0 PL=0
MOVL C01216 V=800.0 PL=0
MOVL C01217 V=800.0 PL=0
MOVL C01218 V=800.0 PL=0
MOVL C01219 V=800.0 PL=0
MOVL C01220 V=800.0 PL=0
MOVL C01221 V=800.0 PL=0
MOVL C01222 V=800.0 PL=0
MOVL C01223 V=800.0 PL=0
MOVL C01224 V=800.0 PL=0
MOVL C01225 V=800.0 PL=0
MOVL C01226 V=800.0 PL=0
MOVL C01227 V=800.0 PL=0
MOVL C01228 V=800.0 PL=0
MOVL C01229 V=800.0 PL=0
MOVL C01230 V=800.0 PL=0
MOVL C01231 V=800.0 PL=0
MOVL C01232 V=800.0 PL=0
MOVL C01233 V=800.0 PL=0
MOVL C01234 V=800.0 PL=0
MOVL C01235 V=800.0 PL=0
MOVL C01236 V=800.0 PL=0
MOVL C01237 V=800.0 PL=0
MOVL C01238 V=800.0 PL=0
MOVL C01239 V=800.0 PL=0
MOVL C01240 V=800.0 PL=0
MOVL C01241 V=800.0 PL=0
MOVL C01242 V=800.0 PL=0
MOVL C01243 V=800.0 PL=0
MOVL C01244 V=800.0 PL=0
MOVL C01245 V=800.0 PL=0
MOVL C01246 V=800.0 PL=0
MOVL C01247 V=800.0 PL=0
MOVL C01248 V=800.0 PL=0
MOVL C01249 V=800.0 PL=0
MOVL C01250 V=800.0 PL=0
MOVL C01251 V=800.0 PL=0
MOVL C01252 V=800.0 PL=0
MOVL C01253 V=800.0 PL=0
MOVL C01254 V=800.0 PL=0
MOVL C01255 V=800.0 PL=0
MOVL C01256 V=800.0 PL=0
MOVL C01257 V=800.0 PL=0
MOVL C01258 V=800.0 PL=0
MOVL C01259 V=800.0 PL=0
MOVL C01260 V=800.0 PL=0
MOVL C01261 V=800.0 PL=0
MOVL C01262 V=800.0 PL=0
MOVL C01263 V=800.0 PL=0
MOVL C01264 V=800.0 PL=0
MOVL C01265 V=800.0 PL=0
MOVL C01266 V=800.0 PL=0
MOVL C01267 V=800.0 PL=0
MOVL C01268 V=800.0 PL=0
MOVL C01269 V=800.0 PL=0
MOVL C01270 V=800.0 PL=0
MOVL C01271 V=800.0 PL=0
MOVL C01272 V=800.0 PL=0
MOVL C01273 V=800.0 PL=0
MOVL C01274 V=800.0 PL=0
MOVL C01275 V=800.0 PL=0
MOVL C01276 V=800.0 PL=0
MOVL C01277 V=800.0 PL=0
MOVL C01278 V=800.0 PL=0
MOVL C01279 V=800.0 PL=0
MOVL C01280 V=800.0 PL=0
MOVL C01281 V=800.0 PL=0
MOVL C01282 V=800.0 PL=0
MOVL C01283 V=800.0 PL=0
MOVL C01284 V=800.0 PL=0
MOVL C01285 V=800.0 PL=0
MOVL C01286 V=800.0 PL=0
MOVL C01287 V=800.0 PL=0
MOVL C01288 V=800.0 PL=0
MOVL C01289 V=800.0 PL=0
MOVL C01290 V=800.0 PL=0
MOVL C01291 V=800.0 PL=0
MOVL C01292 V=800.0 PL=0
MOVL C01293 V=800.0 PL=0
MOVL C01294 V=800.0 PL=0
MOVL C01295 V=800.0 PL=0
MOVL C01296 V=800.0 PL=0
MOVL C01297 V=800.0 PL=0
MOVL C01298 V=800.0 PL=0
MOVL C01299 V=800.0 PL=0
MOVL C01300 V=800.0 PL=0
MOVL C01301 V=800.0 PL=0
MOVL C01302 V=800.0 PL=0
MOVL C01303 V=800.0 PL=0
MOVL C01304 V=800.0 PL=0
MOVL C01305 V=800.0 PL=0
MOVL C01306 V=800.0 PL=0
MOVL C01307 V=800.0 PL=0
MOVL C01308 V=800.0 PL=0
MOVL C01309 V=800.0 PL=0
MOVL C01310 V=800.0 PL=0
MOVL C01311 V=800.0 PL=0
MOVL C01312 V=800.0 PL=0
MOVL C01313 V=800.0 PL=0
MOVL C01314 V=800.0 PL=0
MOVL C01315 V=800.0 PL=0
MOVL C01316 V=800.0 PL=0
MOVL C01317 V=800.0 PL=0
MOVL C01318 V=800.0 PL=0
MOVL C01319 V=800.0 PL=0
MOVL C01320 V=800.0 PL=0
MOVL C01321 V=800.0 PL=0
MOVL C01322 V=800.0 PL=0
MOVL C01323 V=800.0 PL=0
MOVL C01324 V=800.0 PL=0
MOVL C01325 V=800.0 PL=0
MOVL C01326 V=800.0 PL=0
MOVL C01327 V=800.0 PL=0
MOVL C01328 V=800.0 PL=0
MOVL C01329 V=800.0 PL=0
MOVL C01330 V=800.0 PL=0
MOVL C01331 V=800.0 PL=0
MOVL C01332 V=800.0 PL=0
MOVL C01333 V=800.0 PL=0
MOVL C01334 V=800.0 PL=0
MOVL C01335 V=800.0 PL=0
MOVL C01336 V=800.0 PL=0
MOVL C01337 V=800.0 PL=0
MOVL C01338 V=800.0 PL=0
MOVL C01339 V=800.0 PL=0
MOVL C01340 V=800.0 PL=0
MOVL C01341 V=800.0 PL=0
MOVL C01342 V=800.0 PL=0
MOVL C01343 V=800.0 PL=0
MOVL C01344 V=800.0 PL=0
MOVL C01345 V=800.0 PL=0
MOVL C01346 V=800.0 PL=0
MOVL C01347 V=800.0 PL=0
MOVL C01348 V=800.0 PL=0
MOVL C01349 V=800.0 PL=0
MOVL C01350 V=800.0 PL=0
MOVL C01351 V=800.0 PL=0
MOVL C01352 V=800.0 PL=0
MOVL C01353 V=800.0 PL=0
MOVL C01354 V=800.0 PL=0
MOVL C01355 V=800.0 PL=0
MOVL C01356 V=800.0 PL=0
MOVL C01357 V=800.0 PL=0
MOVL C01358 V=800.0 PL=0
MOVL C01359 V=800.0 PL=0
MOVL C01360 V=800.0 PL=0
MOVL C01361 V=800.0 PL=0
MOVL C01362 V=800.0 PL=0
MOVL C01363 V=800.0 PL=0
MOVL C01364 V=800.0 PL=0
MOVL C01365 V=800.0 PL=0
MOVL C01366 V=800.0 PL=0
MOVL C01367 V=800.0 PL=0
MOVL C01368 V=800.0 PL=0
MOVL C01369 V=800.0 PL=0
MOVL C01370 V=800.0 PL=0
MOVL C01371 V=800.0 PL=0
MOVL C01372 V=800.0 PL=0
MOVL C01373 V=800.0 PL=0
MOVL C01374 V=800.0 PL=0
MOVL C01375 V=800.0 PL=0
MOVL C01376 V=800.0 PL=0
MOVL C01377 V=800.0 PL=0
MOVL C01378 V=800.0 PL=0
MOVL C01379 V=800.0 PL=0
MOVL C01380 V=800.0 PL=0
MOVL C01381 V=800.0 PL=0
MOVL C01382 V=800.0 PL=0
MOVL C01383 V=800.0 PL=0
MOVL C01384 V=800.0 PL=0
MOVL C01385 V=800.0 PL=0
MOVL C01386 V=800.0 PL=0
MOVL C01387 V=800.0 PL=0
MOVL C01388 V=800.0 PL=0
MOVL C01389 V=800.0 PL=0
MOVL C01390 V=800.0 PL=0
MOVL C01391 V=800.0 PL=0
MOVL C01392 V=800.0 PL=0
MOVL C01393 V=800.0 PL=0
MOVL C01394 V=800.0 PL=0
MOVL C01395 V=800.0 PL=0
MOVL C01396 V=800.0 PL=0
MOVL C01397 V=800.0 PL=0
MOVL C01398 V=800.0 PL=0
MOVL C01399 V=800.0 PL=0
MOVL C01400 V=800.0 PL=0
MOVL C01401 V=800.0 PL=0
MOVL C01402 V=800.0 PL=0
MOVL C01403 V=800.0 PL=0
MOVL C01404 V=800.0 PL=0
MOVL C01405 V=800.0 PL=0
MOVL C01406 V=800.0 PL=0
MOVL C01407 V=800.0 PL=0
MOVL C01408 V=800.0 PL=0
MOVL C01409 V=800.0 PL=0
MOVL C01410 V=800.0 PL=0
MOVL C01411 V=800.0 PL=0
MOVL C01412 V=800.0 PL=0
MOVL C01413 V=800.0 PL=0
MOVL C01414 V=800.0 PL=0
MOVL C01415 V=800.0 PL=0
MOVL C01416 V=800.0 PL=0
MOVL C01417 V=800.0 PL=0
MOVL C01418 V=800.0 PL=0
MOVL C01419 V=800.0 PL=0
MOVL C01420 V=800.0 PL=0
MOVL C01421 V=800.0 PL=0
MOVL C01422 V=800.0 PL=0
MOVL C01423 V=800.0 PL=0
MOVL C01424 V=800.0 PL=0
MOVL C01425 V=800.0 PL=0
MOVL C01426 V=800.0 PL=0
MOVL C01427 V=800.0 PL=0
MOVL C01428 V=800.0 PL=0
MOVL C01429 V=800.0 PL=0
MOVL C01430 V=800.0 PL=0
MOVL C01431 V=800.0 PL=0
MOVL C01432 V=800.0 PL=0
MOVL C01433 V=800.0 PL=0
MOVL C01434 V=800.0 PL=0
MOVL C01435 V=800.0 PL=0
MOVL C01436 V=800.0 PL=0
MOVL C01437 V=800.0 PL=0
MOVL C01438 V=800.0 PL=0
MOVL C01439 V=800.0 PL=0
MOVL C01440 V=800.0 PL=0
MOVL C01441 V=800.0 PL=0
MOVL C01442 V=800.0 PL=0
MOVL C01443 V=800.0 PL=0
MOVL C01444 V=800.0 PL=0
MOVL C01445 V=800.0 PL=0
MOVL C01446 V=800.0 PL=0
MOVL C01447 V=800.0 PL=0
MOVL C01448 V=800.0 PL=0
MOVL C01449 V=800.0 PL=0
MOVL C01450 V=800.0 PL=0
MOVL C01451 V=800.0 PL=0
MOVL C01452 V=800.0 PL=0
MOVL C01453 V=800.0 PL=0
MOVL C01454 V=800.0 PL=0
MOVL C01455 V=800.0 PL=0
MOVL C01456 V=800.0 PL=0
MOVL C01457 V=800.0 PL=0
MOVL C01458 V=800.0 PL=0
MOVL C01459 V=800.0 PL=0
MOVL C01460 V=800.0 PL=0
MOVL C01461 V=800.0 PL=0
MOVL C01462 V=800.0 PL=0
MOVL C01463 V=800.0 PL=0
MOVL C01464 V=800.0 PL=0
MOVL C01465 V=800.0 PL=0
MOVL C01466 V=800.0 PL=0
MOVL C01467 V=800.0 PL=0
MOVL C01468 V=800.0 PL=0
MOVL C01469 V=800.0 PL=0
MOVL C01470 V=800.0 PL=0
MOVL C01471 V=800.0 PL=0
MOVL C01472 V=800.0 PL=0
MOVL C01473 V=800.0 PL=0
MOVL C01474 V=800.0 PL=0
MOVL C01475 V=800.0 PL=0
MOVL C01476 V=800.0 PL=0
MOVL C01477 V=800.0 PL=0
MOVL C01478 V=800.0 PL=0
MOVL C01479 V=800.0 PL=0
MOVL C01480 V=800.0 PL=0
MOVL C01481 V=800.0 PL=0
MOVL C01482 V=800.0 PL=0
MOVL C01483 V=800.0 PL=0
MOVL C01484 V=800.0 PL=0
MOVL C01485 V=800.0 PL=0
MOVL C01486 V=800.0 PL=0
MOVL C01487 V=800.0 PL=0
MOVL C01488 V=800.0 PL=0
MOVL C01489 V=800.0 PL=0
MOVL C01490 V=800.0 PL=0
MOVL C01491 V=800.0 PL=0
MOVL C01492 V=800.0 PL=0
MOVL C01493 V=800.0 PL=0
MOVL C01494 V=800.0 PL=0
MOVL C01495 V=800.0 PL=0
MOVL C01496 V=800.0 PL=0
MOVL C01497 V=800.0 PL=0
MOVL C01498 V=800.0 PL=0
MOVL C01499 V=800.0 PL=0
MOVL C01500 V=800.0 PL=0
MOVL C01501 V=800.0 PL=0
MOVL C01502 V=800.0 PL=0
MOVL C01503 V=800.0 PL=0
MOVL C01504 V=800.0 PL=0
MOVL C01505 V=800.0 PL=0
MOVL C01506 V=800.0 PL=0
MOVL C01507 V=800.0 PL=0
MOVL C01508 V=800.0 PL=0
MOVL C01509 V=800.0 PL=0
MOVL C01510 V=800.0 PL=0
MOVL C01511 V=800.0 PL=0
MOVL C01512 V=800.0 PL=0
MOVL C01513 V=800.0 PL=0
MOVL C01514 V=800.0 PL=0
MOVL C01515 V=800.0 PL=0
MOVL C01516 V=800.0 PL=0
MOVL C01517 V=800.0 PL=0
MOVL C01518 V=800.0 PL=0
MOVL C01519 V=800.0 PL=0
MOVL C01520 V=800.0 PL=0
MOVL C01521 V=800.0 PL=0
MOVL C01522 V=800.0 PL=0
MOVL C01523 V=800.0 PL=0
MOVL C01524 V=800.0 PL=0
MOVL C01525 V=800.0 PL=0
MOVL C01526 V=800.0 PL=0
MOVL C01527 V=800.0 PL=0
MOVL C01528 V=800.0 PL=0
MOVL C01529 V=800.0 PL=0
MOVL C01530 V=800.0 PL=0
MOVL C01531 V=800.0 PL=0
MOVL C01532 V=800.0 PL=0
MOVL C01533 V=800.0 PL=0
MOVL C01534 V=800.0 PL=0
MOVL C01535 V=800.0 PL=0
MOVL C01536 V=800.0 PL=0
MOVL C01537 V=800.0 PL=0
MOVL C01538 V=800.0 PL=0
MOVL C01539 V=800.0 PL=0
MOVL C01540 V=800.0 PL=0
MOVL C01541 V=800.0 PL=0
MOVL C01542 V=800.0 PL=0
MOVL C01543 V=800.0 PL=0
MOVL C01544 V=800.0 PL=0
MOVL C01545 V=800.0 PL=0
MOVL C01546 V=800.0 PL=0
MOVL C01547 V=800.0 PL=0
MOVL C01548 V=800.0 PL=0
MOVL C01549 V=800.0 PL=0
MOVL C01550 V=800.0 PL=0
MOVL C01551 V=800.0 PL=0
MOVL C01552 V=800.0 PL=0
MOVL C01553 V=800.0 PL=0
MOVL C01554 V=800.0 PL=0
MOVL C01555 V=800.0 PL=0
MOVL C01556 V=800.0 PL=0
MOVL C01557 V=800.0 PL=0
MOVL C01558 V=800.0 PL=0
MOVL C01559 V=800.0 PL=0
MOVL C01560 V=800.0 PL=0
MOVL C01561 V=800.0 PL=0
MOVL C01562 V=800.0 PL=0
MOVL C01563 V=800.0 PL=0
MOVL C01564 V=800.0 PL=0
MOVL C01565 V=800.0 PL=0
MOVL C01566 V=800.0 PL=0
MOVL C01567 V=800.0 PL=0
MOVL C01568 V=800.0 PL=0
MOVL C01569 V=800.0 PL=0
MOVL C01570 V=800.0 PL=0
MOVL C01571 V=800.0 PL=0
MOVL C01572 V=800.0 PL=0
MOVL C01573 V=800.0 PL=0
MOVL C01574 V=800.0 PL=0
MOVL C01575 V=800.0 PL=0
MOVL C01576 V=800.0 PL=0
MOVL C01577 V=800.0 PL=0
MOVL C01578 V=800.0 PL=0
MOVL C01579 V=800.0 PL=0
MOVL C01580 V=800.0 PL=0
MOVL C01581 V=800.0 PL=0
MOVL C01582 V=800.0 PL=0
MOVL C01583 V=800.0 PL=0
MOVL C01584 V=800.0 PL=0
MOVL C01585 V=800.0 PL=0
MOVL C01586 V=800.0 PL=0
MOVL C01587 V=800.0 PL=0
MOVL C01588 V=800.0 PL=0
MOVL C01589 V=800.0 PL=0
MOVL C01590 V=800.0 PL=0
MOVL C01591 V=800.0 PL=0
MOVL C01592 V=800.0 PL=0
MOVL C01593 V=800.0 PL=0
MOVL C01594 V=800.0 PL=0
MOVL C01595 V=800.0 PL=0
MOVL C01596 V=800.0 PL=0
MOVL C01597 V=800.0 PL=0
MOVL C01598 V=800.0 PL=0
MOVL C01599 V=800.0 PL=0
MOVL C01600 V=800.0 PL=0
MOVL C01601 V=800.0 PL=0
MOVL C01602 V=800.0 PL=0
MOVL C01603 V=800.0 PL=0
MOVL C01604 V=800.0 PL=0
MOVL C01605 V=800.0 PL=0
MOVL C01606 V=800.0 PL=0
MOVL C01607 V=800.0 PL=0
MOVL C01608 V=800.0 PL=0
MOVL C01609 V=800.0 PL=0
MOVL C01610 V=800.0 PL=0
MOVL C01611 V=800.0 PL=0
MOVL C01612 V=800.0 PL=0
MOVL C01613 V=800.0 PL=0
MOVL C01614 V=800.0 PL=0
MOVL C01615 V=800.0 PL=0
MOVL C01616 V=800.0 PL=0
MOVL C01617 V=800.0 PL=0
MOVL C01618 V=800.0 PL=0
MOVL C01619 V=800.0 PL=0
MOVL C01620 V=800.0 PL=0
MOVL C01621 V=800.0 PL=0
MOVL C01622 V=800.0 PL=0
MOVL C01623 V=800.0 PL=0
MOVL C01624 V=800.0 PL=0
MOVL C01625 V=800.0 PL=0
MOVL C01626 V=800.0 PL=0
MOVL C01627 V=800.0 PL=0
MOVL C01628 V=800.0 PL=0
MOVL C01629 V=800.0 PL=0
MOVL C01630 V=800.0 PL=0
MOVL C01631 V=800.0 PL=0
MOVL C01632 V=800.0 PL=0
MOVL C01633 V=800.0 PL=0
MOVL C01634 V=800.0 PL=0
MOVL C01635 V=800.0 PL=0
MOVL C01636 V=800.0 PL=0
MOVL C01637 V=800.0 PL=0
MOVL C01638 V=800.0 PL=0
MOVL C01639 V=800.0 PL=0
MOVL C01640 V=800.0 PL=0
MOVL C01641 V=800.0 PL=0
MOVL C01642 V=800.0 PL=0
MOVL C01643 V=800.0 PL=0
MOVL C01644 V=800.0 PL=0
MOVL C01645 V=800.0 PL=0
MOVL C01646 V=800.0 PL=0
MOVL C01647 V=800.0 PL=0
MOVL C01648 V=800.0 PL=0
MOVL C01649 V=800.0 PL=0
MOVL C01650 V=800.0 PL=0
MOVL C01651 V=800.0 PL=0
MOVL C01652 V=800.0 PL=0
MOVL C01653 V=800.0 PL=0
MOVL C01654 V=800.0 PL=0
MOVL C01655 V=800.0 PL=0
MOVL C01656 V=800.0 PL=0
MOVL C01657 V=800.0 PL=0
MOVL C01658 V=800.0 PL=0
MOVL C01659 V=800.0 PL=0
MOVL C01660 V=800.0 PL=0
MOVL C01661 V=800.0 PL=0
MOVL C01662 V=800.0 PL=0
MOVL C01663 V=800.0 PL=0
MOVL C01664 V=800.0 PL=0
MOVL C01665 V=800.0 PL=0
MOVL C01666 V=800.0 PL=0
MOVL C01667 V=800.0 PL=0
MOVL C01668 V=800.0 PL=0
MOVL C01669 V=800.0 PL=0
MOVL C01670 V=800.0 PL=0
MOVL C01671 V=800.0 PL=0
MOVL C01672 V=800.0 PL=0
MOVL C01673 V=800.0 PL=0
MOVL C01674 V=800.0 PL=0
MOVL C01675 V=800.0 PL=0
MOVL C01676 V=800.0 PL=0
MOVL C01677 V=800.0 PL=0
MOVL C01678 V=800.0 PL=0
MOVL C01679 V=800.0 PL=0
MOVL C01680 V=800.0 PL=0
MOVL C01681 V=800.0 PL=0
MOVL C01682 V=800.0 PL=0
MOVL C01683 V=800.0 PL=0
MOVL C01684 V=800.0 PL=0
MOVL C01685 V=800.0 PL=0
MOVL C01686 V=800.0 PL=0
MOVL C01687 V=800.0 PL=0
MOVL C01688 V=800.0 PL=0
MOVL C01689 V=800.0 PL=0
MOVL C01690 V=800.0 PL=0
MOVL C01691 V=800.0 PL=0
MOVL C01692 V=800.0 PL=0
MOVL C01693 V=800.0 PL=0
MOVL C01694 V=800.0 PL=0
MOVL C01695 V=800.0 PL=0
MOVL C01696 V=800.0 PL=0
MOVL C01697 V=800.0 PL=0
MOVL C01698 V=800.0 PL=0
MOVL C01699 V=800.0 PL=0
MOVL C01700 V=800.0 PL=0
MOVL C01701 V=800.0 PL=0
MOVL C01702 V=800.0 PL=0
MOVL C01703 V=800.0 PL=0
MOVL C01704 V=800.0 PL=0
MOVL C01705 V=800.0 PL=0
MOVL C01706 V=800.0 PL=0
MOVL C01707 V=800.0 PL=0
MOVL C01708 V=800.0 PL=0
MOVL C01709 V=800.0 PL=0
MOVL C01710 V=800.0 PL=0
MOVL C01711 V=800.0 PL=0
MOVL C01712 V=800.0 PL=0
MOVL C01713 V=800.0 PL=0
MOVL C01714 V=800.0 PL=0
MOVL C01715 V=800.0 PL=0
MOVL C01716 V=800.0 PL=0
MOVL C01717 V=800.0 PL=0
MOVL C01718 V=800.0 PL=0
MOVL C01719 V=800.0 PL=0
MOVL C01720 V=800.0 PL=0
MOVL C01721 V=800.0 PL=0
MOVL C01722 V=800.0 PL=0
MOVL C01723 V=800.0 PL=0
MOVL C01724 V=800.0 PL=0
MOVL C01725 V=800.0 PL=0
MOVL C01726 V=800.0 PL=0
MOVL C01727 V=800.0 PL=0
MOVL C01728 V=800.0 PL=0
MOVL C01729 V=800.0 PL=0
MOVL C01730 V=800.0 PL=0
MOVL C01731 V=800.0 PL=0
MOVL C01732 V=800.0 PL=0
MOVL C01733 V=800.0 PL=0
MOVL C01734 V=800.0 PL=0
MOVL C01735 V=800.0 PL=0
MOVL C01736 V=800.0 PL=0
MOVL C01737 V=800.0 PL=0
MOVL C01738 V=800.0 PL=0
MOVL C01739 V=800.0 PL=0
MOVL C01740 V=800.0 PL=0
MOVL C01741 V=800.0 PL=0
MOVL C01742 V=800.0 PL=0
MOVL C01743 V=800.0 PL=0
MOVL C01744 V=800.0 PL=0
MOVL C01745 V=800.0 PL=0
MOVL C01746 V=800.0 PL=0
MOVL C01747 V=800.0 PL=0
MOVL C01748 V=800.0 PL=0
MOVL C01749 V=800.0 PL=0
MOVL C01750 V=800.0 PL=0
MOVL C01751 V=800.0 PL=0
MOVL C01752 V=800.0 PL=0
MOVL C01753 V=800.0 PL=0
MOVL C01754 V=800.0 PL=0
MOVL C01755 V=800.0 PL=0
MOVL C01756 V=800.0 PL=0
MOVL C01757 V=800.0 PL=0
MOVL C01758 V=800.0 PL=0
MOVL C01759 V=800.0 PL=0
MOVL C01760 V=800.0 PL=0
MOVL C01761 V=800.0 PL=0
MOVL C01762 V=800.0 PL=0
MOVL C01763 V=800.0 PL=0
MOVL C01764 V=800.0 PL=0
MOVL C01765 V=800.0 PL=0
MOVL C01766 V=800.0 PL=0
MOVL C01767 V=800.0 PL=0
MOVL C01768 V=800.0 PL=0
MOVL C01769 V=800.0 PL=0
MOVL C01770 V=800.0 PL=0
MOVL C01771 V=800.0 PL=0
MOVL C01772 V=800.0 PL=0
MOVL C01773 V=800.0 PL=0
MOVL C01774 V=800.0 PL=0
MOVL C01775 V=800.0 PL=0
MOVL C01776 V=800.0 PL=0
MOVL C01777 V=800.0 PL=0
MOVL C01778 V=800.0 PL=0
MOVL C01779 V=800.0 PL=0
MOVL C01780 V=800.0 PL=0
MOVL C01781 V=800.0 PL=0
MOVL C01782 V=800.0 PL=0
MOVL C01783 V=800.0 PL=0
MOVL C01784 V=800.0 PL=0
MOVL C01785 V=800.0 PL=0
MOVL C01786 V=800.0 PL=0
MOVL C01787 V=800.0 PL=0
MOVL C01788 V=800.0 PL=0
MOVL C01789 V=800.0 PL=0
MOVL C01790 V=800.0 PL=0
MOVL C01791 V=800.0 PL=0
MOVL C01792 V=800.0 PL=0
MOVL C01793 V=800.0 PL=0
MOVL C01794 V=800.0 PL=0
MOVL C01795 V=800.0 PL=0
MOVL C01796 V=800.0 PL=0
MOVL C01797 V=800.0 PL=0
MOVL C01798 V=800.0 PL=0
MOVL C01799 V=800.0 PL=0
MOVL C01800 V=800.0 PL=0
MOVL C01801 V=800.0 PL=0
MOVL C01802 V=800.0 PL=0
MOVL C01803 V=800.0 PL=0
MOVL C01804 V=800.0 PL=0
MOVL C01805 V=800.0 PL=0
MOVL C01806 V=800.0 PL=0
MOVL C01807 V=800.0 PL=0
MOVL C01808 V=800.0 PL=0
MOVL C01809 V=800.0 PL=0
MOVL C01810 V=800.0 PL=0
MOVL C01811 V=800.0 PL=0
MOVL C01812 V=800.0 PL=0
MOVL C01813 V=800.0 PL=0
MOVL C01814 V=800.0 PL=0
MOVL C01815 V=800.0 PL=0
MOVL C01816 V=800.0 PL=0
MOVL C01817 V=800.0 PL=0
MOVL C01818 V=800.0 PL=0
MOVL C01819 V=800.0 PL=0
MOVL C01820 V=800.0 PL=0
MOVL C01821 V=800.0 PL=0
MOVL C01822 V=800.0 PL=0
MOVL C01823 V=800.0 PL=0
MOVL C01824 V=800.0 PL=0
MOVL C01825 V=800.0 PL=0
MOVL C01826 V=800.0 PL=0
MOVL C01827 V=800.0 PL=0
MOVL C01828 V=800.0 PL=0
MOVL C01829 V=800.0 PL=0
MOVL C01830 V=800.0 PL=0
MOVL C01831 V=800.0 PL=0
MOVL C01832 V=800.0 PL=0
MOVL C01833 V=800.0 PL=0
MOVL C01834 V=800.0 PL=0
MOVL C01835 V=800.0 PL=0
MOVL C01836 V=800.0 PL=0
MOVL C01837 V=800.0 PL=0
MOVL C01838 V=800.0 PL=0
MOVL C01839 V=800.0 PL=0
MOVL C01840 V=800.0 PL=0
MOVL C01841 V=800.0 PL=0
MOVL C01842 V=800.0 PL=0
MOVL C01843 V=800.0 PL=0
MOVL C01844 V=800.0 PL=0
MOVL C01845 V=800.0 PL=0
MOVL C01846 V=800.0 PL=0
MOVL C01847 V=800.0 PL=0
MOVL C01848 V=800.0 PL=0
MOVL C01849 V=800.0 PL=0
MOVL C01850 V=800.0 PL=0
MOVL C01851 V=800.0 PL=0
MOVL C01852 V=800.0 PL=0
MOVL C01853 V=800.0 PL=0
MOVL C01854 V=800.0 PL=0
MOVL C01855 V=800.0 PL=0
MOVL C01856 V=800.0 PL=0
MOVL C01857 V=800.0 PL=0
MOVL C01858 V=800.0 PL=0
MOVL C01859 V=800.0 PL=0
MOVL C01860 V=800.0 PL=0
MOVL C01861 V=800.0 PL=0
MOVL C01862 V=800.0 PL=0
MOVL C01863 V=800.0 PL=0
MOVL C01864 V=800.0 PL=0
MOVL C01865 V=800.0 PL=0
MOVL C01866 V=800.0 PL=0
MOVL C01867 V=800.0 PL=0
MOVL C01868 V=800.0 PL=0
MOVL C01869 V=800.0 PL=0
MOVL C01870 V=800.0 PL=0
MOVL C01871 V=800.0 PL=0
MOVL C01872 V=800.0 PL=0
MOVL C01873 V=800.0 PL=0
MOVL C01874 V=800.0 PL=0
MOVL C01875 V=800.0 PL=0
MOVL C01876 V=800.0 PL=0
MOVL C01877 V=800.0 PL=0
MOVL C01878 V=800.0 PL=0
MOVL C01879 V=800.0 PL=0
MOVL C01880 V=800.0 PL=0
MOVL C01881 V=800.0 PL=0
MOVL C01882 V=800.0 PL=0
MOVL C01883 V=800.0 PL=0
MOVL C01884 V=800.0 PL=0
MOVL C01885 V=800.0 PL=0
MOVL C01886 V=800.0 PL=0
MOVL C01887 V=800.0 PL=0
MOVL C01888 V=800.0 PL=0
MOVL C01889 V=800.0 PL=0
MOVL C01890 V=800.0 PL=0
MOVL C01891 V=800.0 PL=0
MOVL C01892 V=800.0 PL=0
MOVL C01893 V=800.0 PL=0
MOVL C01894 V=800.0 PL=0
MOVL C01895 V=800.0 PL=0
MOVL C01896 V=800.0 PL=0
MOVL C01897 V=800.0 PL=0
MOVL C01898 V=800.0 PL=0
MOVL C01899 V=800.0 PL=0
MOVL C01900 V=800.0 PL=0
MOVL C01901 V=800.0 PL=0
MOVL C01902 V=800.0 PL=0
MOVL C01903 V=800.0 PL=0
MOVL C01904 V=800.0 PL=0
MOVL C01905 V=800.0 PL=0
MOVL C01906 V=800.0 PL=0
MOVL C01907 V=800.0 PL=0
MOVL C01908 V=800.0 PL=0
MOVL C01909 V=800.0 PL=0
MOVL C01910 V=800.0 PL=0
MOVL C01911 V=800.0 PL=0
MOVL C01912 V=800.0 PL=0
MOVL C01913 V=800.0 PL=0
MOVL C01914 V=800.0 PL=0
MOVL C01915 V=800.0 PL=0
MOVL C01916 V=800.0 PL=0
MOVL C01917 V=800.0 PL=0
MOVL C01918 V=800.0 PL=0
MOVL C01919 V=800.0 PL=0
MOVL C01920 V=800.0 PL=0
MOVL C01921 V=800.0 PL=0
MOVL C01922 V=800.0 PL=0
MOVL C01923 V=800.0 PL=0
MOVL C01924 V=800.0 PL=0
MOVL C01925 V=800.0 PL=0
MOVL C01926 V=800.0 PL=0
MOVL C01927 V=800.0 PL=0
MOVL C01928 V=800.0 PL=0
MOVL C01929 V=800.0 PL=0
MOVL C01930 V=800.0 PL=0
MOVL C01931 V=800.0 PL=0
MOVL C01932 V=800.0 PL=0
MOVL C01933 V=800.0 PL=0
MOVL C01934 V=800.0 PL=0
MOVL C01935 V=800.0 PL=0
MOVL C01936 V=800.0 PL=0
MOVL C01937 V=800.0 PL=0
MOVL C01938 V=800.0 PL=0
MOVL C01939 V=800.0 PL=0
MOVL C01940 V=800.0 PL=0
MOVL C01941 V=800.0 PL=0
MOVL C01942 V=800.0 PL=0
MOVL C01943 V=800.0 PL=0
MOVL C01944 V=800.0 PL=0
MOVL C01945 V=800.0 PL=0
MOVL C01946 V=800.0 PL=0
MOVL C01947 V=800.0 PL=0
MOVL C01948 V=800.0 PL=0
MOVL C01949 V=800.0 PL=0
MOVL C01950 V=800.0 PL=0
MOVL C01951 V=800.0 PL=0
MOVL C01952 V=800.0 PL=0
MOVL C01953 V=800.0 PL=0
MOVL C01954 V=800.0 PL=0
MOVL C01955 V=800.0 PL=0
MOVL C01956 V=800.0 PL=0
MOVL C01957 V=800.0 PL=0
MOVL C01958 V=800.0 PL=0
MOVL C01959 V=800.0 PL=0
MOVL C01960 V=800.0 PL=0
MOVL C01961 V=800.0 PL=0
MOVL C01962 V=800.0 PL=0
MOVL C01963 V=800.0 PL=0
MOVL C01964 V=800.0 PL=0
MOVL C01965 V=800.0 PL=0
MOVL C01966 V=800.0 PL=0
MOVL C01967 V=800.0 PL=0
MOVL C01968 V=800.0 PL=0
MOVL C01969 V=800.0 PL=0
MOVL C01970 V=800.0 PL=0
MOVL C01971 V=800.0 PL=0
MOVL C01972 V=800.0 PL=0
MOVL C01973 V=800.0 PL=0
MOVL C01974 V=800.0 PL=0
MOVL C01975 V=800.0 PL=0
MOVL C01976 V=800.0 PL=0
MOVL C01977 V=800.0 PL=0
MOVL C01978 V=800.0 PL=0
MOVL C01979 V=800.0 PL=0
MOVL C01980 V=800.0 PL=0
MOVL C01981 V=800.0 PL=0
MOVL C01982 V=800.0 PL=0
MOVL C01983 V=800.0 PL=0
MOVL C01984 V=800.0 PL=0
MOVL C01985 V=800.0 PL=0
MOVL C01986 V=800.0 PL=0
MOVL C01987 V=800.0 PL=0
MOVL C01988 V=800.0 PL=0
MOVL C01989 V=800.0 PL=0
MOVL C01990 V=800.0 PL=0
MOVL C01991 V=800.0 PL=0
MOVL C01992 V=800.0 PL=0
MOVL C01993 V=800.0 PL=0
MOVL C01994 V=800.0 PL=0
MOVL C01995 V=800.0 PL=0
MOVL C01996 V=800.0 PL=0
MOVL C01997 V=800.0 PL=0
MOVL C01998 V=800.0 PL=0
MOVL C01999 V=800.0 PL=0
MOVL C02000 V=800.0 PL=0
